DATA_BLOCK "InstCycleTimerDataset1"   // DB63
TITLE = Instanz CycleTimerDataset1 / Instance CycleTimerDataset1
{ DB_Accessible_From_OPC_UA := 'FALSE' }
AUTHOR : SICAR
FAMILY : ProdData
// Instanz DB / Instance DB
// stored: DBAccessibleFromOPCUA false, InstanceOfName LSicar_ProdDataCycleTimer, InstanceOfType FB
"LSicar_ProdDataCycleTimer"
   // VAR_INPUT
   //    numberConfigDataSets { ExternalAccessible := 'False'; ExternalVisible := 'False'; ExternalWritable := 'False'} : Int := 0;
   //    dataSetNumber { ExternalAccessible := 'False'; ExternalVisible := 'False'; ExternalWritable := 'False'} : UInt := 0;
   //    pulse100ms { ExternalAccessible := 'False'; ExternalVisible := 'False'; ExternalWritable := 'False'} : Bool := FALSE;
   // END_VAR
   // VAR_IN_OUT
   //    numberOfDataSets : "LSicar_typeNumberOfDataSets";
   //    dataSet : "LSicar_typeCycleTimer";
   // END_VAR
   // VAR
   //    statCycleTimer { ExternalAccessible := 'False'; ExternalVisible := 'False'; ExternalWritable := 'False'} : Array[0..20] of "LSicar_typeCycleTimerStruct";
   //    statRisEdgeResetAllExt { ExternalAccessible := 'False'; ExternalVisible := 'False'; ExternalWritable := 'False'} : Bool := FALSE;
   //    statPosPulseResetAllExt { ExternalAccessible := 'False'; ExternalVisible := 'False'; ExternalWritable := 'False'} : Bool := FALSE;
   //    statRisEdgeResetAll { ExternalAccessible := 'False'; ExternalVisible := 'False'; ExternalWritable := 'False'} : Bool := FALSE;
   //    statPosPulseResetAll { ExternalAccessible := 'False'; ExternalVisible := 'False'; ExternalWritable := 'False'} : Bool := FALSE;
   // END_VAR
BEGIN
   statCycleTimer[0..20].falEdgeRun := FALSE;
   statCycleTimer[0..20].negPulseRun := FALSE;
   statCycleTimer[0..20].risEdgeReset := FALSE;
   statCycleTimer[0..20].posPulseReset := FALSE;
   statCycleTimer[0..20].operateValue := 0;
END_DATA_BLOCK

DATA_BLOCK "InstCycleTimerDataset2"   // DB79
TITLE = Instanz CycleTimerDataset2 / Instance CycleTimerDataset2
{ DB_Accessible_From_OPC_UA := 'FALSE' }
AUTHOR : SICAR
FAMILY : ProdData
// Instanz DB / Instance DB
// stored: DBAccessibleFromOPCUA false, InstanceOfName LSicar_ProdDataCycleTimer, InstanceOfType FB
"LSicar_ProdDataCycleTimer"
   // VAR_INPUT
   //    numberConfigDataSets { ExternalAccessible := 'False'; ExternalVisible := 'False'; ExternalWritable := 'False'} : Int := 0;
   //    dataSetNumber { ExternalAccessible := 'False'; ExternalVisible := 'False'; ExternalWritable := 'False'} : UInt := 0;
   //    pulse100ms { ExternalAccessible := 'False'; ExternalVisible := 'False'; ExternalWritable := 'False'} : Bool := FALSE;
   // END_VAR
   // VAR_IN_OUT
   //    numberOfDataSets : "LSicar_typeNumberOfDataSets";
   //    dataSet : "LSicar_typeCycleTimer";
   // END_VAR
   // VAR
   //    statCycleTimer { ExternalAccessible := 'False'; ExternalVisible := 'False'; ExternalWritable := 'False'} : Array[0..20] of "LSicar_typeCycleTimerStruct";
   //    statRisEdgeResetAllExt { ExternalAccessible := 'False'; ExternalVisible := 'False'; ExternalWritable := 'False'} : Bool := FALSE;
   //    statPosPulseResetAllExt { ExternalAccessible := 'False'; ExternalVisible := 'False'; ExternalWritable := 'False'} : Bool := FALSE;
   //    statRisEdgeResetAll { ExternalAccessible := 'False'; ExternalVisible := 'False'; ExternalWritable := 'False'} : Bool := FALSE;
   //    statPosPulseResetAll { ExternalAccessible := 'False'; ExternalVisible := 'False'; ExternalWritable := 'False'} : Bool := FALSE;
   // END_VAR
BEGIN
   statCycleTimer[0..20].falEdgeRun := FALSE;
   statCycleTimer[0..20].negPulseRun := FALSE;
   statCycleTimer[0..20].risEdgeReset := FALSE;
   statCycleTimer[0..20].posPulseReset := FALSE;
   statCycleTimer[0..20].operateValue := 0;
END_DATA_BLOCK

DATA_BLOCK "InstCycleTimerDataset3"   // DB114
AUTHOR : SICAR
FAMILY : ProdData
VERSION : 1.0
// stored: InstanceOfName LSicar_ProdDataCycleTimer, InstanceOfType FB
"LSicar_ProdDataCycleTimer"
   // VAR_INPUT
   //    numberConfigDataSets { ExternalAccessible := 'False'; ExternalVisible := 'False'; ExternalWritable := 'False'} : Int;
   //    dataSetNumber { ExternalAccessible := 'False'; ExternalVisible := 'False'; ExternalWritable := 'False'} : UInt;
   //    pulse100ms { ExternalAccessible := 'False'; ExternalVisible := 'False'; ExternalWritable := 'False'} : Bool;
   // END_VAR
   // VAR_IN_OUT
   //    numberOfDataSets : "LSicar_typeNumberOfDataSets";
   //    dataSet : "LSicar_typeCycleTimer";
   // END_VAR
   // VAR
   //    statCycleTimer { ExternalAccessible := 'False'; ExternalVisible := 'False'; ExternalWritable := 'False'} : Array[0..20] of "LSicar_typeCycleTimerStruct";
   //    statRisEdgeResetAllExt { ExternalAccessible := 'False'; ExternalVisible := 'False'; ExternalWritable := 'False'} : Bool;
   //    statPosPulseResetAllExt { ExternalAccessible := 'False'; ExternalVisible := 'False'; ExternalWritable := 'False'} : Bool;
   //    statRisEdgeResetAll { ExternalAccessible := 'False'; ExternalVisible := 'False'; ExternalWritable := 'False'} : Bool;
   //    statPosPulseResetAll { ExternalAccessible := 'False'; ExternalVisible := 'False'; ExternalWritable := 'False'} : Bool;
   // END_VAR
BEGIN
END_DATA_BLOCK

DATA_BLOCK "InstCycleTimerDataset4"   // DB494
AUTHOR : SICAR
FAMILY : ProdData
VERSION : 1.0
// stored: InstanceOfName LSicar_ProdDataCycleTimer, InstanceOfType FB
"LSicar_ProdDataCycleTimer"
   // VAR_INPUT
   //    numberConfigDataSets { ExternalAccessible := 'False'; ExternalVisible := 'False'; ExternalWritable := 'False'} : Int;
   //    dataSetNumber { ExternalAccessible := 'False'; ExternalVisible := 'False'; ExternalWritable := 'False'} : UInt;
   //    pulse100ms { ExternalAccessible := 'False'; ExternalVisible := 'False'; ExternalWritable := 'False'} : Bool;
   // END_VAR
   // VAR_IN_OUT
   //    numberOfDataSets : "LSicar_typeNumberOfDataSets";
   //    dataSet : "LSicar_typeCycleTimer";
   // END_VAR
   // VAR
   //    statCycleTimer { ExternalAccessible := 'False'; ExternalVisible := 'False'; ExternalWritable := 'False'} : Array[0..20] of "LSicar_typeCycleTimerStruct";
   //    statRisEdgeResetAllExt { ExternalAccessible := 'False'; ExternalVisible := 'False'; ExternalWritable := 'False'} : Bool;
   //    statPosPulseResetAllExt { ExternalAccessible := 'False'; ExternalVisible := 'False'; ExternalWritable := 'False'} : Bool;
   //    statRisEdgeResetAll { ExternalAccessible := 'False'; ExternalVisible := 'False'; ExternalWritable := 'False'} : Bool;
   //    statPosPulseResetAll { ExternalAccessible := 'False'; ExternalVisible := 'False'; ExternalWritable := 'False'} : Bool;
   // END_VAR
BEGIN
END_DATA_BLOCK

DATA_BLOCK "InstCycleTimerDataset5"   // DB216
AUTHOR : SICAR
FAMILY : ProdData
VERSION : 1.0
// stored: InstanceOfName LSicar_ProdDataCycleTimer, InstanceOfType FB
"LSicar_ProdDataCycleTimer"
   // VAR_INPUT
   //    numberConfigDataSets { ExternalAccessible := 'False'; ExternalVisible := 'False'; ExternalWritable := 'False'} : Int;
   //    dataSetNumber { ExternalAccessible := 'False'; ExternalVisible := 'False'; ExternalWritable := 'False'} : UInt;
   //    pulse100ms { ExternalAccessible := 'False'; ExternalVisible := 'False'; ExternalWritable := 'False'} : Bool;
   // END_VAR
   // VAR_IN_OUT
   //    numberOfDataSets : "LSicar_typeNumberOfDataSets";
   //    dataSet : "LSicar_typeCycleTimer";
   // END_VAR
   // VAR
   //    statCycleTimer { ExternalAccessible := 'False'; ExternalVisible := 'False'; ExternalWritable := 'False'} : Array[0..20] of "LSicar_typeCycleTimerStruct";
   //    statRisEdgeResetAllExt { ExternalAccessible := 'False'; ExternalVisible := 'False'; ExternalWritable := 'False'} : Bool;
   //    statPosPulseResetAllExt { ExternalAccessible := 'False'; ExternalVisible := 'False'; ExternalWritable := 'False'} : Bool;
   //    statRisEdgeResetAll { ExternalAccessible := 'False'; ExternalVisible := 'False'; ExternalWritable := 'False'} : Bool;
   //    statPosPulseResetAll { ExternalAccessible := 'False'; ExternalVisible := 'False'; ExternalWritable := 'False'} : Bool;
   // END_VAR
BEGIN
END_DATA_BLOCK

DATA_BLOCK "InstCycleTimerDataset6"   // DB258
AUTHOR : SICAR
FAMILY : ProdData
VERSION : 1.0
// stored: InstanceOfName LSicar_ProdDataCycleTimer, InstanceOfType FB
"LSicar_ProdDataCycleTimer"
   // VAR_INPUT
   //    numberConfigDataSets { ExternalAccessible := 'False'; ExternalVisible := 'False'; ExternalWritable := 'False'} : Int;
   //    dataSetNumber { ExternalAccessible := 'False'; ExternalVisible := 'False'; ExternalWritable := 'False'} : UInt;
   //    pulse100ms { ExternalAccessible := 'False'; ExternalVisible := 'False'; ExternalWritable := 'False'} : Bool;
   // END_VAR
   // VAR_IN_OUT
   //    numberOfDataSets : "LSicar_typeNumberOfDataSets";
   //    dataSet : "LSicar_typeCycleTimer";
   // END_VAR
   // VAR
   //    statCycleTimer { ExternalAccessible := 'False'; ExternalVisible := 'False'; ExternalWritable := 'False'} : Array[0..20] of "LSicar_typeCycleTimerStruct";
   //    statRisEdgeResetAllExt { ExternalAccessible := 'False'; ExternalVisible := 'False'; ExternalWritable := 'False'} : Bool;
   //    statPosPulseResetAllExt { ExternalAccessible := 'False'; ExternalVisible := 'False'; ExternalWritable := 'False'} : Bool;
   //    statRisEdgeResetAll { ExternalAccessible := 'False'; ExternalVisible := 'False'; ExternalWritable := 'False'} : Bool;
   //    statPosPulseResetAll { ExternalAccessible := 'False'; ExternalVisible := 'False'; ExternalWritable := 'False'} : Bool;
   // END_VAR
BEGIN
END_DATA_BLOCK

DATA_BLOCK "InstCycleTimerDataset7"   // DB264
AUTHOR : SICAR
FAMILY : ProdData
VERSION : 1.0
// stored: InstanceOfName LSicar_ProdDataCycleTimer, InstanceOfType FB
"LSicar_ProdDataCycleTimer"
   // VAR_INPUT
   //    numberConfigDataSets { ExternalAccessible := 'False'; ExternalVisible := 'False'; ExternalWritable := 'False'} : Int;
   //    dataSetNumber { ExternalAccessible := 'False'; ExternalVisible := 'False'; ExternalWritable := 'False'} : UInt;
   //    pulse100ms { ExternalAccessible := 'False'; ExternalVisible := 'False'; ExternalWritable := 'False'} : Bool;
   // END_VAR
   // VAR_IN_OUT
   //    numberOfDataSets : "LSicar_typeNumberOfDataSets";
   //    dataSet : "LSicar_typeCycleTimer";
   // END_VAR
   // VAR
   //    statCycleTimer { ExternalAccessible := 'False'; ExternalVisible := 'False'; ExternalWritable := 'False'} : Array[0..20] of "LSicar_typeCycleTimerStruct";
   //    statRisEdgeResetAllExt { ExternalAccessible := 'False'; ExternalVisible := 'False'; ExternalWritable := 'False'} : Bool;
   //    statPosPulseResetAllExt { ExternalAccessible := 'False'; ExternalVisible := 'False'; ExternalWritable := 'False'} : Bool;
   //    statRisEdgeResetAll { ExternalAccessible := 'False'; ExternalVisible := 'False'; ExternalWritable := 'False'} : Bool;
   //    statPosPulseResetAll { ExternalAccessible := 'False'; ExternalVisible := 'False'; ExternalWritable := 'False'} : Bool;
   // END_VAR
BEGIN
END_DATA_BLOCK

DATA_BLOCK "InstCycleTimerDataset8"   // DB267
AUTHOR : SICAR
FAMILY : ProdData
VERSION : 1.0
// stored: InstanceOfName LSicar_ProdDataCycleTimer, InstanceOfType FB
"LSicar_ProdDataCycleTimer"
   // VAR_INPUT
   //    numberConfigDataSets { ExternalAccessible := 'False'; ExternalVisible := 'False'; ExternalWritable := 'False'} : Int;
   //    dataSetNumber { ExternalAccessible := 'False'; ExternalVisible := 'False'; ExternalWritable := 'False'} : UInt;
   //    pulse100ms { ExternalAccessible := 'False'; ExternalVisible := 'False'; ExternalWritable := 'False'} : Bool;
   // END_VAR
   // VAR_IN_OUT
   //    numberOfDataSets : "LSicar_typeNumberOfDataSets";
   //    dataSet : "LSicar_typeCycleTimer";
   // END_VAR
   // VAR
   //    statCycleTimer { ExternalAccessible := 'False'; ExternalVisible := 'False'; ExternalWritable := 'False'} : Array[0..20] of "LSicar_typeCycleTimerStruct";
   //    statRisEdgeResetAllExt { ExternalAccessible := 'False'; ExternalVisible := 'False'; ExternalWritable := 'False'} : Bool;
   //    statPosPulseResetAllExt { ExternalAccessible := 'False'; ExternalVisible := 'False'; ExternalWritable := 'False'} : Bool;
   //    statRisEdgeResetAll { ExternalAccessible := 'False'; ExternalVisible := 'False'; ExternalWritable := 'False'} : Bool;
   //    statPosPulseResetAll { ExternalAccessible := 'False'; ExternalVisible := 'False'; ExternalWritable := 'False'} : Bool;
   // END_VAR
BEGIN
END_DATA_BLOCK

DATA_BLOCK "InstLimitValueDataset1"   // DB54
TITLE = Instanz LimitValueDataset1 / Instance LimitValueDataset1
{ DB_Accessible_From_OPC_UA := 'FALSE' }
AUTHOR : SICAR
FAMILY : ProdData
// Instanz DB / Instance DB
// stored: DBAccessibleFromOPCUA false, InstanceOfName LSicar_ProdDataLimitValues, InstanceOfType FB
"LSicar_ProdDataLimitValues"
   // VAR_INPUT
   //    numberConfigDataSets { ExternalAccessible := 'False'; ExternalVisible := 'False'; ExternalWritable := 'False'} : Int := 0;
   //    dataSetNumber { ExternalAccessible := 'False'; ExternalVisible := 'False'; ExternalWritable := 'False'} : UInt := 0;
   // END_VAR
   // VAR_IN_OUT
   //    numberOfDataSets : "LSicar_typeNumberOfDataSets";
   //    dataSet : "LSicar_typeLimitValue";
   //    colorCodeSelectButton { ExternalAccessible := 'False'; ExternalVisible := 'False'; ExternalWritable := 'False'} : UInt := 0;
   // END_VAR
   // VAR
   //    statLimitValue { ExternalAccessible := 'False'; ExternalVisible := 'False'; ExternalWritable := 'False'} : Array[0..10] of "LSicar_typeEdgePulseStruct";
   //    statPrewarnActive { ExternalAccessible := 'False'; ExternalVisible := 'False'; ExternalWritable := 'False'} : Bool := FALSE;
   //    statAlarmActive { ExternalAccessible := 'False'; ExternalVisible := 'False'; ExternalWritable := 'False'} : Bool := FALSE;
   // END_VAR
BEGIN
   statLimitValue[0..10].risEdgeCountUp := FALSE;
   statLimitValue[0..10].posPulseCountUp := FALSE;
   statLimitValue[0..10].risEdgeCountDown := FALSE;
   statLimitValue[0..10].posPulseCountDown := FALSE;
   statLimitValue[0..10].risEdgeReset := FALSE;
   statLimitValue[0..10].posPulseReset := FALSE;
END_DATA_BLOCK

DATA_BLOCK "InstLimitValueDataset2"   // DB55
TITLE = Instanz LimitValueDataset2 / Instance LimitValueDataset2
{ DB_Accessible_From_OPC_UA := 'FALSE' }
AUTHOR : SICAR
FAMILY : ProdData
// Instanz DB / Instance DB
// stored: DBAccessibleFromOPCUA false, InstanceOfName LSicar_ProdDataLimitValues, InstanceOfType FB
"LSicar_ProdDataLimitValues"
   // VAR_INPUT
   //    numberConfigDataSets { ExternalAccessible := 'False'; ExternalVisible := 'False'; ExternalWritable := 'False'} : Int := 0;
   //    dataSetNumber { ExternalAccessible := 'False'; ExternalVisible := 'False'; ExternalWritable := 'False'} : UInt := 0;
   // END_VAR
   // VAR_IN_OUT
   //    numberOfDataSets : "LSicar_typeNumberOfDataSets";
   //    dataSet : "LSicar_typeLimitValue";
   //    colorCodeSelectButton { ExternalAccessible := 'False'; ExternalVisible := 'False'; ExternalWritable := 'False'} : UInt := 0;
   // END_VAR
   // VAR
   //    statLimitValue { ExternalAccessible := 'False'; ExternalVisible := 'False'; ExternalWritable := 'False'} : Array[0..10] of "LSicar_typeEdgePulseStruct";
   //    statPrewarnActive { ExternalAccessible := 'False'; ExternalVisible := 'False'; ExternalWritable := 'False'} : Bool := FALSE;
   //    statAlarmActive { ExternalAccessible := 'False'; ExternalVisible := 'False'; ExternalWritable := 'False'} : Bool := FALSE;
   // END_VAR
BEGIN
   statLimitValue[0..10].risEdgeCountUp := FALSE;
   statLimitValue[0..10].posPulseCountUp := FALSE;
   statLimitValue[0..10].risEdgeCountDown := FALSE;
   statLimitValue[0..10].posPulseCountDown := FALSE;
   statLimitValue[0..10].risEdgeReset := FALSE;
   statLimitValue[0..10].posPulseReset := FALSE;
END_DATA_BLOCK

DATA_BLOCK "InstShiftCounterDataset1"   // DB62
TITLE = Instanz ShiftCounterDataset1 / Instance ShiftCounterDataset1
{ DB_Accessible_From_OPC_UA := 'FALSE' }
AUTHOR : SICAR
FAMILY : ProdData
// Instanz DB / Instance DB
// stored: DBAccessibleFromOPCUA false, InstanceOfName LSicar_ProdDataShiftCounter, InstanceOfType FB
"LSicar_ProdDataShiftCounter"
   // VAR_INPUT
   //    numberConfigDataSets { ExternalAccessible := 'False'; ExternalVisible := 'False'; ExternalWritable := 'False'} : Int := 0;
   //    dataSetNumber { ExternalAccessible := 'False'; ExternalVisible := 'False'; ExternalWritable := 'False'} : UInt := 0;
   // END_VAR
   // VAR_IN_OUT
   //    numberOfDataSets : "LSicar_typeNumberOfDataSets";
   //    dataSet : "LSicar_typeShiftCounter";
   // END_VAR
   // VAR
   //    statPartsCurrentCount { ExternalAccessible := 'False'; ExternalVisible := 'False'; ExternalWritable := 'False'} : Array[0..10] of "LSicar_typeEdgePulseStruct";
   //    statRisEdgeResetAllExt { ExternalAccessible := 'False'; ExternalVisible := 'False'; ExternalWritable := 'False'} : Bool := FALSE;
   //    statPosPulseResetAllExt { ExternalAccessible := 'False'; ExternalVisible := 'False'; ExternalWritable := 'False'} : Bool := FALSE;
   //    statRisEdgeResetAll { ExternalAccessible := 'False'; ExternalVisible := 'False'; ExternalWritable := 'False'} : Bool := FALSE;
   //    statPosPulseResetAll { ExternalAccessible := 'False'; ExternalVisible := 'False'; ExternalWritable := 'False'} : Bool := FALSE;
   // END_VAR
BEGIN
   statPartsCurrentCount[0..10].risEdgeCountUp := FALSE;
   statPartsCurrentCount[0..10].posPulseCountUp := FALSE;
   statPartsCurrentCount[0..10].risEdgeCountDown := FALSE;
   statPartsCurrentCount[0..10].posPulseCountDown := FALSE;
   statPartsCurrentCount[0..10].risEdgeReset := FALSE;
   statPartsCurrentCount[0..10].posPulseReset := FALSE;
END_DATA_BLOCK

DATA_BLOCK "InstShiftCounterDataset2"   // DB64
TITLE = Instanz ShiftCounterDataset2 / Instance ShiftCounterDataset2
{ DB_Accessible_From_OPC_UA := 'FALSE' }
AUTHOR : SICAR
FAMILY : ProdData
// Instanz DB / Instance DB
// stored: DBAccessibleFromOPCUA false, InstanceOfName LSicar_ProdDataShiftCounter, InstanceOfType FB
"LSicar_ProdDataShiftCounter"
   // VAR_INPUT
   //    numberConfigDataSets { ExternalAccessible := 'False'; ExternalVisible := 'False'; ExternalWritable := 'False'} : Int := 0;
   //    dataSetNumber { ExternalAccessible := 'False'; ExternalVisible := 'False'; ExternalWritable := 'False'} : UInt := 0;
   // END_VAR
   // VAR_IN_OUT
   //    numberOfDataSets : "LSicar_typeNumberOfDataSets";
   //    dataSet : "LSicar_typeShiftCounter";
   // END_VAR
   // VAR
   //    statPartsCurrentCount { ExternalAccessible := 'False'; ExternalVisible := 'False'; ExternalWritable := 'False'} : Array[0..10] of "LSicar_typeEdgePulseStruct";
   //    statRisEdgeResetAllExt { ExternalAccessible := 'False'; ExternalVisible := 'False'; ExternalWritable := 'False'} : Bool := FALSE;
   //    statPosPulseResetAllExt { ExternalAccessible := 'False'; ExternalVisible := 'False'; ExternalWritable := 'False'} : Bool := FALSE;
   //    statRisEdgeResetAll { ExternalAccessible := 'False'; ExternalVisible := 'False'; ExternalWritable := 'False'} : Bool := FALSE;
   //    statPosPulseResetAll { ExternalAccessible := 'False'; ExternalVisible := 'False'; ExternalWritable := 'False'} : Bool := FALSE;
   // END_VAR
BEGIN
   statPartsCurrentCount[0..10].risEdgeCountUp := FALSE;
   statPartsCurrentCount[0..10].posPulseCountUp := FALSE;
   statPartsCurrentCount[0..10].risEdgeCountDown := FALSE;
   statPartsCurrentCount[0..10].posPulseCountDown := FALSE;
   statPartsCurrentCount[0..10].risEdgeReset := FALSE;
   statPartsCurrentCount[0..10].posPulseReset := FALSE;
END_DATA_BLOCK

DATA_BLOCK "InstShiftCounterOeeDset1"   // DB124
TITLE = Instanz ShiftCounterOeeDset1 / Instance ShiftCounterOeeDset1
{ DB_Accessible_From_OPC_UA := 'FALSE' }
AUTHOR : SICAR
FAMILY : ProdData
// Instanz DB / Instance DB
// stored: DBAccessibleFromOPCUA false, InstanceOfName LSicar_ProdDataShiftCounterOee, InstanceOfType FB
"LSicar_ProdDataShiftCounterOee"
   // VAR_INPUT
   //    numberConfigDataSets { ExternalAccessible := 'False'; ExternalVisible := 'False'; ExternalWritable := 'False'} : Int := 0;
   //    dataSetNumber { ExternalAccessible := 'False'; ExternalVisible := 'False'; ExternalWritable := 'False'} : UInt := 0;
   //    shiftProdTimeTarget { ExternalAccessible := 'False'; ExternalVisible := 'False'; ExternalWritable := 'False'} : Time := T#0MS;
   //    shiftProdTimeExpired { ExternalAccessible := 'False'; ExternalVisible := 'False'; ExternalWritable := 'False'} : Time := T#0MS;
   // END_VAR
   // VAR_IN_OUT
   //    numberOfDataSets : "LSicar_typeNumberOfDataSets";
   //    dataSet : "LSicar_typeShiftCounterOee";
   // END_VAR
   // VAR
   //    statPartsCurrentCount { ExternalAccessible := 'False'; ExternalVisible := 'False'; ExternalWritable := 'False'} : Array[0..10] of "LSicar_typeEdgePulseStruct";
   //    statPartsCurrentCountOk { ExternalAccessible := 'False'; ExternalVisible := 'False'; ExternalWritable := 'False'} : Array[0..10] of "LSicar_typeEdgePulseStruct";
   //    statFactor { ExternalAccessible := 'False'; ExternalVisible := 'False'; ExternalWritable := 'False'} : "LSicar_typeFactorOee";
   //    statTimeFactorTrend { ExternalAccessible := 'False'; ExternalVisible := 'False'; ExternalWritable := 'False'} : Real := 0.0;
   //    statShiftProdTimeTarget { ExternalAccessible := 'False'; ExternalVisible := 'False'; ExternalWritable := 'False'} : Real := 0.0;
   //    statShiftProdTimeExpired { ExternalAccessible := 'False'; ExternalVisible := 'False'; ExternalWritable := 'False'} : Real := 0.0;
   //    statRisEdgeResetAllExt { ExternalAccessible := 'False'; ExternalVisible := 'False'; ExternalWritable := 'False'} : Bool := FALSE;
   //    statPosPulseResetAllExt { ExternalAccessible := 'False'; ExternalVisible := 'False'; ExternalWritable := 'False'} : Bool := FALSE;
   //    statRisEdgeResetAll { ExternalAccessible := 'False'; ExternalVisible := 'False'; ExternalWritable := 'False'} : Bool := FALSE;
   //    statPosPulseResetAll { ExternalAccessible := 'False'; ExternalVisible := 'False'; ExternalWritable := 'False'} : Bool := FALSE;
   // END_VAR
BEGIN
   statPartsCurrentCount[0..10].risEdgeCountUp := FALSE;
   statPartsCurrentCount[0..10].posPulseCountUp := FALSE;
   statPartsCurrentCount[0..10].risEdgeCountDown := FALSE;
   statPartsCurrentCount[0..10].posPulseCountDown := FALSE;
   statPartsCurrentCount[0..10].risEdgeReset := FALSE;
   statPartsCurrentCount[0..10].posPulseReset := FALSE;
   statPartsCurrentCountOk[0..10].risEdgeCountUp := FALSE;
   statPartsCurrentCountOk[0..10].posPulseCountUp := FALSE;
   statPartsCurrentCountOk[0..10].risEdgeCountDown := FALSE;
   statPartsCurrentCountOk[0..10].posPulseCountDown := FALSE;
   statPartsCurrentCountOk[0..10].risEdgeReset := FALSE;
   statPartsCurrentCountOk[0..10].posPulseReset := FALSE;
   statFactor.utilization := 0.0;
   statFactor.efficiency := 0.0;
   statFactor.quality := 0.0;
END_DATA_BLOCK

DATA_BLOCK "InstShiftCounterOeeDset2"   // DB125
TITLE = Instanz ShiftCounterOeeDset2 / Instance ShiftCounterOeeDset2
{ DB_Accessible_From_OPC_UA := 'FALSE' }
AUTHOR : SICAR
FAMILY : ProdData
// Instanz DB / Instance DB
// stored: DBAccessibleFromOPCUA false, InstanceOfName LSicar_ProdDataShiftCounterOee, InstanceOfType FB
"LSicar_ProdDataShiftCounterOee"
   // VAR_INPUT
   //    numberConfigDataSets { ExternalAccessible := 'False'; ExternalVisible := 'False'; ExternalWritable := 'False'} : Int := 0;
   //    dataSetNumber { ExternalAccessible := 'False'; ExternalVisible := 'False'; ExternalWritable := 'False'} : UInt := 0;
   //    shiftProdTimeTarget { ExternalAccessible := 'False'; ExternalVisible := 'False'; ExternalWritable := 'False'} : Time := T#0MS;
   //    shiftProdTimeExpired { ExternalAccessible := 'False'; ExternalVisible := 'False'; ExternalWritable := 'False'} : Time := T#0MS;
   // END_VAR
   // VAR_IN_OUT
   //    numberOfDataSets : "LSicar_typeNumberOfDataSets";
   //    dataSet : "LSicar_typeShiftCounterOee";
   // END_VAR
   // VAR
   //    statPartsCurrentCount { ExternalAccessible := 'False'; ExternalVisible := 'False'; ExternalWritable := 'False'} : Array[0..10] of "LSicar_typeEdgePulseStruct";
   //    statPartsCurrentCountOk { ExternalAccessible := 'False'; ExternalVisible := 'False'; ExternalWritable := 'False'} : Array[0..10] of "LSicar_typeEdgePulseStruct";
   //    statFactor { ExternalAccessible := 'False'; ExternalVisible := 'False'; ExternalWritable := 'False'} : "LSicar_typeFactorOee";
   //    statTimeFactorTrend { ExternalAccessible := 'False'; ExternalVisible := 'False'; ExternalWritable := 'False'} : Real := 0.0;
   //    statShiftProdTimeTarget { ExternalAccessible := 'False'; ExternalVisible := 'False'; ExternalWritable := 'False'} : Real := 0.0;
   //    statShiftProdTimeExpired { ExternalAccessible := 'False'; ExternalVisible := 'False'; ExternalWritable := 'False'} : Real := 0.0;
   //    statRisEdgeResetAllExt { ExternalAccessible := 'False'; ExternalVisible := 'False'; ExternalWritable := 'False'} : Bool := FALSE;
   //    statPosPulseResetAllExt { ExternalAccessible := 'False'; ExternalVisible := 'False'; ExternalWritable := 'False'} : Bool := FALSE;
   //    statRisEdgeResetAll { ExternalAccessible := 'False'; ExternalVisible := 'False'; ExternalWritable := 'False'} : Bool := FALSE;
   //    statPosPulseResetAll { ExternalAccessible := 'False'; ExternalVisible := 'False'; ExternalWritable := 'False'} : Bool := FALSE;
   // END_VAR
BEGIN
   statPartsCurrentCount[0..10].risEdgeCountUp := FALSE;
   statPartsCurrentCount[0..10].posPulseCountUp := FALSE;
   statPartsCurrentCount[0..10].risEdgeCountDown := FALSE;
   statPartsCurrentCount[0..10].posPulseCountDown := FALSE;
   statPartsCurrentCount[0..10].risEdgeReset := FALSE;
   statPartsCurrentCount[0..10].posPulseReset := FALSE;
   statPartsCurrentCountOk[0..10].risEdgeCountUp := FALSE;
   statPartsCurrentCountOk[0..10].posPulseCountUp := FALSE;
   statPartsCurrentCountOk[0..10].risEdgeCountDown := FALSE;
   statPartsCurrentCountOk[0..10].posPulseCountDown := FALSE;
   statPartsCurrentCountOk[0..10].risEdgeReset := FALSE;
   statPartsCurrentCountOk[0..10].posPulseReset := FALSE;
   statFactor.utilization := 0.0;
   statFactor.efficiency := 0.0;
   statFactor.quality := 0.0;
END_DATA_BLOCK

DATA_BLOCK "InstShiftProductionTimes"   // DB113
TITLE = Instance ShiftProductionTimes
{ DB_Accessible_From_OPC_UA := 'FALSE' }
AUTHOR : SICAR
FAMILY : Shift
// Instance DB
// stored: DBAccessibleFromOPCUA false, InstanceOfName LSicar_ShiftProductionTimes, InstanceOfType FB
"LSicar_ShiftProductionTimes"
   // VAR_OUTPUT
   //    shiftProdTimeTarget { ExternalAccessible := 'False'; ExternalVisible := 'False'; ExternalWritable := 'False'} : Time := T#0MS;
   //    shiftProdTimeExpired { ExternalAccessible := 'False'; ExternalVisible := 'False'; ExternalWritable := 'False'} : Time := T#0MS;
   //    shiftActive { ExternalAccessible := 'False'; ExternalVisible := 'False'; ExternalWritable := 'False'} : Bool := FALSE;
   //    shiftFinishedPulse { ExternalAccessible := 'False'; ExternalVisible := 'False'; ExternalWritable := 'False'} : Bool := FALSE;
   // END_VAR
   // VAR_IN_OUT
   //    dateAndTime : "LSicar_typeGlobalDateTime";
   //    prodTimesHmi : "LSicar_typeProdTimesHmi";
   // END_VAR
   // VAR
   //    statCurrShiftTimes { ExternalAccessible := 'False'; ExternalVisible := 'False'; ExternalWritable := 'False'} : "LSicar_typeShiftTimes1Shift";
   //    statActual { ExternalAccessible := 'False'; ExternalVisible := 'False'; ExternalWritable := 'False'} : Time_Of_Day := TOD#00:00:00;
   //    statBefore { ExternalAccessible := 'False'; ExternalVisible := 'False'; ExternalWritable := 'False'} : Time_Of_Day := TOD#00:00:00;
   //    statDayChange { ExternalAccessible := 'False'; ExternalVisible := 'False'; ExternalWritable := 'False'} : Bool := FALSE;
   //    statDayChangeSet { ExternalAccessible := 'False'; ExternalVisible := 'False'; ExternalWritable := 'False'} : Bool := FALSE;
   //    statShift { ExternalAccessible := 'False'; ExternalVisible := 'False'; ExternalWritable := 'False'} : "LSicar_typeShiftmodelInfo";
   //    statProdTimeExpired { ExternalAccessible := 'False'; ExternalVisible := 'False'; ExternalWritable := 'False'} : Time := T#0MS;
   //    statBreak { ExternalAccessible := 'False'; ExternalVisible := 'False'; ExternalWritable := 'False'} : Array[0..4] of "LSicar_typeShiftmodelInfo";
   //    statBreakDurationSummary { ExternalAccessible := 'False'; ExternalVisible := 'False'; ExternalWritable := 'False'} : Time := T#0MS;
   //    statBreakActiveSummary { ExternalAccessible := 'False'; ExternalVisible := 'False'; ExternalWritable := 'False'} : Bool := FALSE;
   //    statBreakCount { ExternalAccessible := 'False'; ExternalVisible := 'False'; ExternalWritable := 'False'} : USInt := 0;
   //    statProdTimeExpired1 { ExternalAccessible := 'False'; ExternalVisible := 'False'; ExternalWritable := 'False'} : Time := T#0MS;
   //    statProdTimeExpired2 { ExternalAccessible := 'False'; ExternalVisible := 'False'; ExternalWritable := 'False'} : Time := T#0MS;
   //    statFalEdgeShiftActive { ExternalAccessible := 'False'; ExternalVisible := 'False'; ExternalWritable := 'False'} : Bool := FALSE;
   //    statNegPulseShiftActive { ExternalAccessible := 'False'; ExternalVisible := 'False'; ExternalWritable := 'False'} : Bool := FALSE;
   // END_VAR
BEGIN
   statCurrShiftTimes.start := TOD#00:00:00;
   statCurrShiftTimes.break[0..4].start := TOD#00:00:00;
   statCurrShiftTimes.break[0..4].startCircuitTime := TOD#00:00:00;
   statCurrShiftTimes.break[0..4].endCircuitTime := TOD#00:00:00;
   statCurrShiftTimes.break[0..4].end := TOD#00:00:00;
   statCurrShiftTimes.end := TOD#00:00:00;
   statShift.configured := FALSE;
   statShift.active := FALSE;
   statShift.duration := T#0MS;
   statBreak[0..4].configured := FALSE;
   statBreak[0..4].active := FALSE;
   statBreak[0..4].duration := T#0MS;
END_DATA_BLOCK

DATA_BLOCK "InstShiftmodel"   // DB101
TITLE = Instanz Shiftmodel / InstanceShiftmodel
{ DB_Accessible_From_OPC_UA := 'FALSE' }
AUTHOR : SICAR
FAMILY : Shiftmodel
// Instanz DB / Instance DB
// stored: DBAccessibleFromOPCUA false, InstanceOfName LSicar_Shiftmodel, InstanceOfType FB
"LSicar_Shiftmodel"
   // VAR_OUTPUT
   //    currentShiftCircuitTimes { ExternalAccessible := 'False'; ExternalVisible := 'False'; ExternalWritable := 'False'} : "LSicar_typeShiftmodTime1Shift";
   //    currentShiftTimes { ExternalAccessible := 'False'; ExternalVisible := 'False'; ExternalWritable := 'False'} : "LSicar_typeShiftTimes1Shift";
   // END_VAR
   // VAR_IN_OUT
   //    dateAndTime : "LSicar_typeGlobalDateTime";
   //    shiftTimesHmi : "LSicar_typeShiftmodelHmi";
   //    shiftTimesList : Array[0..10] of "LSicar_typeShiftmodTime1DaySel";
   // END_VAR
   // VAR
   //    statListIdx { ExternalAccessible := 'False'; ExternalVisible := 'False'; ExternalWritable := 'False'} : DInt := 0;
   //    statHmiTimesDay { ExternalAccessible := 'False'; ExternalVisible := 'False'; ExternalWritable := 'False'} : Array[0..7] of "LSicar_typeShiftmodTime1Day";
   //    statHmiSignalsDay { ExternalAccessible := 'False'; ExternalVisible := 'False'; ExternalWritable := 'False'} : Array[0..7] of "LSicar_typeShiftmodSign1Day";
   //    statHmiActualDay { ExternalAccessible := 'False'; ExternalVisible := 'False'; ExternalWritable := 'False'} : USInt := 0;
   //    statShiftTimesListOn { ExternalAccessible := 'False'; ExternalVisible := 'False'; ExternalWritable := 'False'} : Bool := FALSE;
   //    statSummaryHmi { ExternalAccessible := 'False'; ExternalVisible := 'False'; ExternalWritable := 'False'} : "LSicar_typeShiftmodSumHmi";
   //    statHmiShiftmoListindex { ExternalAccessible := 'False'; ExternalVisible := 'False'; ExternalWritable := 'False'} : USInt := 1;
   //    statZeroDay { ExternalAccessible := 'False'; ExternalVisible := 'False'; ExternalWritable := 'False'} : "LSicar_typeShiftmodTime1Day";
   //    statListIndexOld { ExternalAccessible := 'False'; ExternalVisible := 'False'; ExternalWritable := 'False'} : DInt := 1;
   //    statNumberOfWorkDays { ExternalAccessible := 'False'; ExternalVisible := 'False'; ExternalWritable := 'False'} : USInt := 0;
   //    statTimeOfDayActual { ExternalAccessible := 'False'; ExternalVisible := 'False'; ExternalWritable := 'False'} : Time_Of_Day := TOD#00:00:00;
   //    statShiftActual { ExternalAccessible := 'False'; ExternalVisible := 'False'; ExternalWritable := 'False'} : USInt := 0;
   //    statDayCount { ExternalAccessible := 'False'; ExternalVisible := 'False'; ExternalWritable := 'False'} : USInt := 1;
   //    statBreakCount { ExternalAccessible := 'False'; ExternalVisible := 'False'; ExternalWritable := 'False'} : USInt := 0;
   //    statDayChangeNightShift { ExternalAccessible := 'False'; ExternalVisible := 'False'; ExternalWritable := 'False'} : Bool := FALSE;
   //    statDayChangeCircuitTime { ExternalAccessible := 'False'; ExternalVisible := 'False'; ExternalWritable := 'False'} : Bool := FALSE;
   //    statCheckCircuitTime { ExternalAccessible := 'False'; ExternalVisible := 'False'; ExternalWritable := 'False'} : "LSicar_typeShiftCircuitTimes";
   //    statRisEdge { ExternalAccessible := 'False'; ExternalVisible := 'False'; ExternalWritable := 'False'} : "LSicar_typeShiftmodSumHmi";
   //    statPosPulse { ExternalAccessible := 'False'; ExternalVisible := 'False'; ExternalWritable := 'False'} : "LSicar_typeShiftmodSumHmi";
   //    statFalEdge { ExternalAccessible := 'False'; ExternalVisible := 'False'; ExternalWritable := 'False'} : "LSicar_typeShiftmodSumHmi";
   //    statNegPulse { ExternalAccessible := 'False'; ExternalVisible := 'False'; ExternalWritable := 'False'} : "LSicar_typeShiftmodSumHmi";
   //    statTimesAndCircuit { ExternalAccessible := 'False'; ExternalVisible := 'False'; ExternalWritable := 'False'} : "LSicar_typeShiftmodTime1Shift";
   //    statOnlyTimes { ExternalAccessible := 'False'; ExternalVisible := 'False'; ExternalWritable := 'False'} : "LSicar_typeShiftTimes1Shift";
   //    statRisEdgeListOn { ExternalAccessible := 'False'; ExternalVisible := 'False'; ExternalWritable := 'False'} : Bool := FALSE;
   //    statPosPulseListOn { ExternalAccessible := 'False'; ExternalVisible := 'False'; ExternalWritable := 'False'} : Bool := FALSE;
   //    statFalEdgeListOn { ExternalAccessible := 'False'; ExternalVisible := 'False'; ExternalWritable := 'False'} : Bool := FALSE;
   //    statNegPulseListOn { ExternalAccessible := 'False'; ExternalVisible := 'False'; ExternalWritable := 'False'} : Bool := FALSE;
   //    statRisEdgeListChange { ExternalAccessible := 'False'; ExternalVisible := 'False'; ExternalWritable := 'False'} : Bool := FALSE;
   //    statPosPulseListChange { ExternalAccessible := 'False'; ExternalVisible := 'False'; ExternalWritable := 'False'} : Bool := FALSE;
   //    statFirstCycle { ExternalAccessible := 'False'; ExternalVisible := 'False'; ExternalWritable := 'False'} : Bool := TRUE;
   // END_VAR
BEGIN
   currentShiftCircuitTimes.endCircuitTime := TOD#00:00:00;
   currentShiftCircuitTimes.start := TOD#00:00:00;
   currentShiftCircuitTimes.break[0..4].start := TOD#00:00:00;
   currentShiftCircuitTimes.break[0..4].startCircuitTime := TOD#00:00:00;
   currentShiftCircuitTimes.break[0..4].endCircuitTime := TOD#00:00:00;
   currentShiftCircuitTimes.break[0..4].end := TOD#00:00:00;
   currentShiftCircuitTimes.end := TOD#00:00:00;
   currentShiftCircuitTimes.startCircuitTime := TOD#00:00:00;
   currentShiftTimes.start := TOD#00:00:00;
   currentShiftTimes.break[0..4].start := TOD#00:00:00;
   currentShiftTimes.break[0..4].startCircuitTime := TOD#00:00:00;
   currentShiftTimes.break[0..4].endCircuitTime := TOD#00:00:00;
   currentShiftTimes.break[0..4].end := TOD#00:00:00;
   currentShiftTimes.end := TOD#00:00:00;
   statHmiTimesDay[0].shift[0..3].endCircuitTime := TOD#00:00:00;
   statHmiTimesDay[1].shift[0..3].endCircuitTime := TOD#00:00:00;
   statHmiTimesDay[2].shift[0..3].endCircuitTime := TOD#00:00:00;
   statHmiTimesDay[3].shift[0..3].endCircuitTime := TOD#00:00:00;
   statHmiTimesDay[4].shift[0..3].endCircuitTime := TOD#00:00:00;
   statHmiTimesDay[5].shift[0..3].endCircuitTime := TOD#00:00:00;
   statHmiTimesDay[6].shift[0..3].endCircuitTime := TOD#00:00:00;
   statHmiTimesDay[7].shift[0..3].endCircuitTime := TOD#00:00:00;
   statHmiTimesDay[0].shift[0..3].start := TOD#00:00:00;
   statHmiTimesDay[1].shift[0..3].start := TOD#00:00:00;
   statHmiTimesDay[2].shift[0..3].start := TOD#00:00:00;
   statHmiTimesDay[3].shift[0..3].start := TOD#00:00:00;
   statHmiTimesDay[4].shift[0..3].start := TOD#00:00:00;
   statHmiTimesDay[5].shift[0..3].start := TOD#00:00:00;
   statHmiTimesDay[6].shift[0..3].start := TOD#00:00:00;
   statHmiTimesDay[7].shift[0..3].start := TOD#00:00:00;
   statHmiTimesDay[0].shift[0].break[0..4].start := TOD#00:00:00;
   statHmiTimesDay[0].shift[1].break[0..4].start := TOD#00:00:00;
   statHmiTimesDay[0].shift[2].break[0..4].start := TOD#00:00:00;
   statHmiTimesDay[0].shift[3].break[0..4].start := TOD#00:00:00;
   statHmiTimesDay[1].shift[0].break[0..4].start := TOD#00:00:00;
   statHmiTimesDay[1].shift[1].break[0..4].start := TOD#00:00:00;
   statHmiTimesDay[1].shift[2].break[0..4].start := TOD#00:00:00;
   statHmiTimesDay[1].shift[3].break[0..4].start := TOD#00:00:00;
   statHmiTimesDay[2].shift[0].break[0..4].start := TOD#00:00:00;
   statHmiTimesDay[2].shift[1].break[0..4].start := TOD#00:00:00;
   statHmiTimesDay[2].shift[2].break[0..4].start := TOD#00:00:00;
   statHmiTimesDay[2].shift[3].break[0..4].start := TOD#00:00:00;
   statHmiTimesDay[3].shift[0].break[0..4].start := TOD#00:00:00;
   statHmiTimesDay[3].shift[1].break[0..4].start := TOD#00:00:00;
   statHmiTimesDay[3].shift[2].break[0..4].start := TOD#00:00:00;
   statHmiTimesDay[3].shift[3].break[0..4].start := TOD#00:00:00;
   statHmiTimesDay[4].shift[0].break[0..4].start := TOD#00:00:00;
   statHmiTimesDay[4].shift[1].break[0..4].start := TOD#00:00:00;
   statHmiTimesDay[4].shift[2].break[0..4].start := TOD#00:00:00;
   statHmiTimesDay[4].shift[3].break[0..4].start := TOD#00:00:00;
   statHmiTimesDay[5].shift[0].break[0..4].start := TOD#00:00:00;
   statHmiTimesDay[5].shift[1].break[0..4].start := TOD#00:00:00;
   statHmiTimesDay[5].shift[2].break[0..4].start := TOD#00:00:00;
   statHmiTimesDay[5].shift[3].break[0..4].start := TOD#00:00:00;
   statHmiTimesDay[6].shift[0].break[0..4].start := TOD#00:00:00;
   statHmiTimesDay[6].shift[1].break[0..4].start := TOD#00:00:00;
   statHmiTimesDay[6].shift[2].break[0..4].start := TOD#00:00:00;
   statHmiTimesDay[6].shift[3].break[0..4].start := TOD#00:00:00;
   statHmiTimesDay[7].shift[0].break[0..4].start := TOD#00:00:00;
   statHmiTimesDay[7].shift[1].break[0..4].start := TOD#00:00:00;
   statHmiTimesDay[7].shift[2].break[0..4].start := TOD#00:00:00;
   statHmiTimesDay[7].shift[3].break[0..4].start := TOD#00:00:00;
   statHmiTimesDay[0].shift[0].break[0..4].startCircuitTime := TOD#00:00:00;
   statHmiTimesDay[0].shift[1].break[0..4].startCircuitTime := TOD#00:00:00;
   statHmiTimesDay[0].shift[2].break[0..4].startCircuitTime := TOD#00:00:00;
   statHmiTimesDay[0].shift[3].break[0..4].startCircuitTime := TOD#00:00:00;
   statHmiTimesDay[1].shift[0].break[0..4].startCircuitTime := TOD#00:00:00;
   statHmiTimesDay[1].shift[1].break[0..4].startCircuitTime := TOD#00:00:00;
   statHmiTimesDay[1].shift[2].break[0..4].startCircuitTime := TOD#00:00:00;
   statHmiTimesDay[1].shift[3].break[0..4].startCircuitTime := TOD#00:00:00;
   statHmiTimesDay[2].shift[0].break[0..4].startCircuitTime := TOD#00:00:00;
   statHmiTimesDay[2].shift[1].break[0..4].startCircuitTime := TOD#00:00:00;
   statHmiTimesDay[2].shift[2].break[0..4].startCircuitTime := TOD#00:00:00;
   statHmiTimesDay[2].shift[3].break[0..4].startCircuitTime := TOD#00:00:00;
   statHmiTimesDay[3].shift[0].break[0..4].startCircuitTime := TOD#00:00:00;
   statHmiTimesDay[3].shift[1].break[0..4].startCircuitTime := TOD#00:00:00;
   statHmiTimesDay[3].shift[2].break[0..4].startCircuitTime := TOD#00:00:00;
   statHmiTimesDay[3].shift[3].break[0..4].startCircuitTime := TOD#00:00:00;
   statHmiTimesDay[4].shift[0].break[0..4].startCircuitTime := TOD#00:00:00;
   statHmiTimesDay[4].shift[1].break[0..4].startCircuitTime := TOD#00:00:00;
   statHmiTimesDay[4].shift[2].break[0..4].startCircuitTime := TOD#00:00:00;
   statHmiTimesDay[4].shift[3].break[0..4].startCircuitTime := TOD#00:00:00;
   statHmiTimesDay[5].shift[0].break[0..4].startCircuitTime := TOD#00:00:00;
   statHmiTimesDay[5].shift[1].break[0..4].startCircuitTime := TOD#00:00:00;
   statHmiTimesDay[5].shift[2].break[0..4].startCircuitTime := TOD#00:00:00;
   statHmiTimesDay[5].shift[3].break[0..4].startCircuitTime := TOD#00:00:00;
   statHmiTimesDay[6].shift[0].break[0..4].startCircuitTime := TOD#00:00:00;
   statHmiTimesDay[6].shift[1].break[0..4].startCircuitTime := TOD#00:00:00;
   statHmiTimesDay[6].shift[2].break[0..4].startCircuitTime := TOD#00:00:00;
   statHmiTimesDay[6].shift[3].break[0..4].startCircuitTime := TOD#00:00:00;
   statHmiTimesDay[7].shift[0].break[0..4].startCircuitTime := TOD#00:00:00;
   statHmiTimesDay[7].shift[1].break[0..4].startCircuitTime := TOD#00:00:00;
   statHmiTimesDay[7].shift[2].break[0..4].startCircuitTime := TOD#00:00:00;
   statHmiTimesDay[7].shift[3].break[0..4].startCircuitTime := TOD#00:00:00;
   statHmiTimesDay[0].shift[0].break[0..4].endCircuitTime := TOD#00:00:00;
   statHmiTimesDay[0].shift[1].break[0..4].endCircuitTime := TOD#00:00:00;
   statHmiTimesDay[0].shift[2].break[0..4].endCircuitTime := TOD#00:00:00;
   statHmiTimesDay[0].shift[3].break[0..4].endCircuitTime := TOD#00:00:00;
   statHmiTimesDay[1].shift[0].break[0..4].endCircuitTime := TOD#00:00:00;
   statHmiTimesDay[1].shift[1].break[0..4].endCircuitTime := TOD#00:00:00;
   statHmiTimesDay[1].shift[2].break[0..4].endCircuitTime := TOD#00:00:00;
   statHmiTimesDay[1].shift[3].break[0..4].endCircuitTime := TOD#00:00:00;
   statHmiTimesDay[2].shift[0].break[0..4].endCircuitTime := TOD#00:00:00;
   statHmiTimesDay[2].shift[1].break[0..4].endCircuitTime := TOD#00:00:00;
   statHmiTimesDay[2].shift[2].break[0..4].endCircuitTime := TOD#00:00:00;
   statHmiTimesDay[2].shift[3].break[0..4].endCircuitTime := TOD#00:00:00;
   statHmiTimesDay[3].shift[0].break[0..4].endCircuitTime := TOD#00:00:00;
   statHmiTimesDay[3].shift[1].break[0..4].endCircuitTime := TOD#00:00:00;
   statHmiTimesDay[3].shift[2].break[0..4].endCircuitTime := TOD#00:00:00;
   statHmiTimesDay[3].shift[3].break[0..4].endCircuitTime := TOD#00:00:00;
   statHmiTimesDay[4].shift[0].break[0..4].endCircuitTime := TOD#00:00:00;
   statHmiTimesDay[4].shift[1].break[0..4].endCircuitTime := TOD#00:00:00;
   statHmiTimesDay[4].shift[2].break[0..4].endCircuitTime := TOD#00:00:00;
   statHmiTimesDay[4].shift[3].break[0..4].endCircuitTime := TOD#00:00:00;
   statHmiTimesDay[5].shift[0].break[0..4].endCircuitTime := TOD#00:00:00;
   statHmiTimesDay[5].shift[1].break[0..4].endCircuitTime := TOD#00:00:00;
   statHmiTimesDay[5].shift[2].break[0..4].endCircuitTime := TOD#00:00:00;
   statHmiTimesDay[5].shift[3].break[0..4].endCircuitTime := TOD#00:00:00;
   statHmiTimesDay[6].shift[0].break[0..4].endCircuitTime := TOD#00:00:00;
   statHmiTimesDay[6].shift[1].break[0..4].endCircuitTime := TOD#00:00:00;
   statHmiTimesDay[6].shift[2].break[0..4].endCircuitTime := TOD#00:00:00;
   statHmiTimesDay[6].shift[3].break[0..4].endCircuitTime := TOD#00:00:00;
   statHmiTimesDay[7].shift[0].break[0..4].endCircuitTime := TOD#00:00:00;
   statHmiTimesDay[7].shift[1].break[0..4].endCircuitTime := TOD#00:00:00;
   statHmiTimesDay[7].shift[2].break[0..4].endCircuitTime := TOD#00:00:00;
   statHmiTimesDay[7].shift[3].break[0..4].endCircuitTime := TOD#00:00:00;
   statHmiTimesDay[0].shift[0].break[0..4].end := TOD#00:00:00;
   statHmiTimesDay[0].shift[1].break[0..4].end := TOD#00:00:00;
   statHmiTimesDay[0].shift[2].break[0..4].end := TOD#00:00:00;
   statHmiTimesDay[0].shift[3].break[0..4].end := TOD#00:00:00;
   statHmiTimesDay[1].shift[0].break[0..4].end := TOD#00:00:00;
   statHmiTimesDay[1].shift[1].break[0..4].end := TOD#00:00:00;
   statHmiTimesDay[1].shift[2].break[0..4].end := TOD#00:00:00;
   statHmiTimesDay[1].shift[3].break[0..4].end := TOD#00:00:00;
   statHmiTimesDay[2].shift[0].break[0..4].end := TOD#00:00:00;
   statHmiTimesDay[2].shift[1].break[0..4].end := TOD#00:00:00;
   statHmiTimesDay[2].shift[2].break[0..4].end := TOD#00:00:00;
   statHmiTimesDay[2].shift[3].break[0..4].end := TOD#00:00:00;
   statHmiTimesDay[3].shift[0].break[0..4].end := TOD#00:00:00;
   statHmiTimesDay[3].shift[1].break[0..4].end := TOD#00:00:00;
   statHmiTimesDay[3].shift[2].break[0..4].end := TOD#00:00:00;
   statHmiTimesDay[3].shift[3].break[0..4].end := TOD#00:00:00;
   statHmiTimesDay[4].shift[0].break[0..4].end := TOD#00:00:00;
   statHmiTimesDay[4].shift[1].break[0..4].end := TOD#00:00:00;
   statHmiTimesDay[4].shift[2].break[0..4].end := TOD#00:00:00;
   statHmiTimesDay[4].shift[3].break[0..4].end := TOD#00:00:00;
   statHmiTimesDay[5].shift[0].break[0..4].end := TOD#00:00:00;
   statHmiTimesDay[5].shift[1].break[0..4].end := TOD#00:00:00;
   statHmiTimesDay[5].shift[2].break[0..4].end := TOD#00:00:00;
   statHmiTimesDay[5].shift[3].break[0..4].end := TOD#00:00:00;
   statHmiTimesDay[6].shift[0].break[0..4].end := TOD#00:00:00;
   statHmiTimesDay[6].shift[1].break[0..4].end := TOD#00:00:00;
   statHmiTimesDay[6].shift[2].break[0..4].end := TOD#00:00:00;
   statHmiTimesDay[6].shift[3].break[0..4].end := TOD#00:00:00;
   statHmiTimesDay[7].shift[0].break[0..4].end := TOD#00:00:00;
   statHmiTimesDay[7].shift[1].break[0..4].end := TOD#00:00:00;
   statHmiTimesDay[7].shift[2].break[0..4].end := TOD#00:00:00;
   statHmiTimesDay[7].shift[3].break[0..4].end := TOD#00:00:00;
   statHmiTimesDay[0].shift[0..3].end := TOD#00:00:00;
   statHmiTimesDay[1].shift[0..3].end := TOD#00:00:00;
   statHmiTimesDay[2].shift[0..3].end := TOD#00:00:00;
   statHmiTimesDay[3].shift[0..3].end := TOD#00:00:00;
   statHmiTimesDay[4].shift[0..3].end := TOD#00:00:00;
   statHmiTimesDay[5].shift[0..3].end := TOD#00:00:00;
   statHmiTimesDay[6].shift[0..3].end := TOD#00:00:00;
   statHmiTimesDay[7].shift[0..3].end := TOD#00:00:00;
   statHmiTimesDay[0].shift[0..3].startCircuitTime := TOD#00:00:00;
   statHmiTimesDay[1].shift[0..3].startCircuitTime := TOD#00:00:00;
   statHmiTimesDay[2].shift[0..3].startCircuitTime := TOD#00:00:00;
   statHmiTimesDay[3].shift[0..3].startCircuitTime := TOD#00:00:00;
   statHmiTimesDay[4].shift[0..3].startCircuitTime := TOD#00:00:00;
   statHmiTimesDay[5].shift[0..3].startCircuitTime := TOD#00:00:00;
   statHmiTimesDay[6].shift[0..3].startCircuitTime := TOD#00:00:00;
   statHmiTimesDay[7].shift[0..3].startCircuitTime := TOD#00:00:00;
   statHmiSignalsDay[0].shift[0..3].shiftConfig := FALSE;
   statHmiSignalsDay[1].shift[0..3].shiftConfig := FALSE;
   statHmiSignalsDay[2].shift[0..3].shiftConfig := FALSE;
   statHmiSignalsDay[3].shift[0..3].shiftConfig := FALSE;
   statHmiSignalsDay[4].shift[0..3].shiftConfig := FALSE;
   statHmiSignalsDay[5].shift[0..3].shiftConfig := FALSE;
   statHmiSignalsDay[6].shift[0..3].shiftConfig := FALSE;
   statHmiSignalsDay[7].shift[0..3].shiftConfig := FALSE;
   statHmiSignalsDay[0].shift[0..3].shiftActive := FALSE;
   statHmiSignalsDay[1].shift[0..3].shiftActive := FALSE;
   statHmiSignalsDay[2].shift[0..3].shiftActive := FALSE;
   statHmiSignalsDay[3].shift[0..3].shiftActive := FALSE;
   statHmiSignalsDay[4].shift[0..3].shiftActive := FALSE;
   statHmiSignalsDay[5].shift[0..3].shiftActive := FALSE;
   statHmiSignalsDay[6].shift[0..3].shiftActive := FALSE;
   statHmiSignalsDay[7].shift[0..3].shiftActive := FALSE;
   statHmiSignalsDay[0].shift[0..3].shiftEndCirTimeConfig := FALSE;
   statHmiSignalsDay[1].shift[0..3].shiftEndCirTimeConfig := FALSE;
   statHmiSignalsDay[2].shift[0..3].shiftEndCirTimeConfig := FALSE;
   statHmiSignalsDay[3].shift[0..3].shiftEndCirTimeConfig := FALSE;
   statHmiSignalsDay[4].shift[0..3].shiftEndCirTimeConfig := FALSE;
   statHmiSignalsDay[5].shift[0..3].shiftEndCirTimeConfig := FALSE;
   statHmiSignalsDay[6].shift[0..3].shiftEndCirTimeConfig := FALSE;
   statHmiSignalsDay[7].shift[0..3].shiftEndCirTimeConfig := FALSE;
   statHmiSignalsDay[0].shift[0..3].shiftStartCirTimeConfig := FALSE;
   statHmiSignalsDay[1].shift[0..3].shiftStartCirTimeConfig := FALSE;
   statHmiSignalsDay[2].shift[0..3].shiftStartCirTimeConfig := FALSE;
   statHmiSignalsDay[3].shift[0..3].shiftStartCirTimeConfig := FALSE;
   statHmiSignalsDay[4].shift[0..3].shiftStartCirTimeConfig := FALSE;
   statHmiSignalsDay[5].shift[0..3].shiftStartCirTimeConfig := FALSE;
   statHmiSignalsDay[6].shift[0..3].shiftStartCirTimeConfig := FALSE;
   statHmiSignalsDay[7].shift[0..3].shiftStartCirTimeConfig := FALSE;
   statHmiSignalsDay[0].shift[0..3].shiftEndCirTimeActive := FALSE;
   statHmiSignalsDay[1].shift[0..3].shiftEndCirTimeActive := FALSE;
   statHmiSignalsDay[2].shift[0..3].shiftEndCirTimeActive := FALSE;
   statHmiSignalsDay[3].shift[0..3].shiftEndCirTimeActive := FALSE;
   statHmiSignalsDay[4].shift[0..3].shiftEndCirTimeActive := FALSE;
   statHmiSignalsDay[5].shift[0..3].shiftEndCirTimeActive := FALSE;
   statHmiSignalsDay[6].shift[0..3].shiftEndCirTimeActive := FALSE;
   statHmiSignalsDay[7].shift[0..3].shiftEndCirTimeActive := FALSE;
   statHmiSignalsDay[0].shift[0..3].shiftStartCirTimeActive := FALSE;
   statHmiSignalsDay[1].shift[0..3].shiftStartCirTimeActive := FALSE;
   statHmiSignalsDay[2].shift[0..3].shiftStartCirTimeActive := FALSE;
   statHmiSignalsDay[3].shift[0..3].shiftStartCirTimeActive := FALSE;
   statHmiSignalsDay[4].shift[0..3].shiftStartCirTimeActive := FALSE;
   statHmiSignalsDay[5].shift[0..3].shiftStartCirTimeActive := FALSE;
   statHmiSignalsDay[6].shift[0..3].shiftStartCirTimeActive := FALSE;
   statHmiSignalsDay[7].shift[0..3].shiftStartCirTimeActive := FALSE;
   statHmiSignalsDay[0].shift[0..3].shiftSignalsHmi := 16#00;
   statHmiSignalsDay[1].shift[0..3].shiftSignalsHmi := 16#00;
   statHmiSignalsDay[2].shift[0..3].shiftSignalsHmi := 16#00;
   statHmiSignalsDay[3].shift[0..3].shiftSignalsHmi := 16#00;
   statHmiSignalsDay[4].shift[0..3].shiftSignalsHmi := 16#00;
   statHmiSignalsDay[5].shift[0..3].shiftSignalsHmi := 16#00;
   statHmiSignalsDay[6].shift[0..3].shiftSignalsHmi := 16#00;
   statHmiSignalsDay[7].shift[0..3].shiftSignalsHmi := 16#00;
   statHmiSignalsDay[0].shift[0].break[0..4].config := FALSE;
   statHmiSignalsDay[0].shift[1].break[0..4].config := FALSE;
   statHmiSignalsDay[0].shift[2].break[0..4].config := FALSE;
   statHmiSignalsDay[0].shift[3].break[0..4].config := FALSE;
   statHmiSignalsDay[1].shift[0].break[0..4].config := FALSE;
   statHmiSignalsDay[1].shift[1].break[0..4].config := FALSE;
   statHmiSignalsDay[1].shift[2].break[0..4].config := FALSE;
   statHmiSignalsDay[1].shift[3].break[0..4].config := FALSE;
   statHmiSignalsDay[2].shift[0].break[0..4].config := FALSE;
   statHmiSignalsDay[2].shift[1].break[0..4].config := FALSE;
   statHmiSignalsDay[2].shift[2].break[0..4].config := FALSE;
   statHmiSignalsDay[2].shift[3].break[0..4].config := FALSE;
   statHmiSignalsDay[3].shift[0].break[0..4].config := FALSE;
   statHmiSignalsDay[3].shift[1].break[0..4].config := FALSE;
   statHmiSignalsDay[3].shift[2].break[0..4].config := FALSE;
   statHmiSignalsDay[3].shift[3].break[0..4].config := FALSE;
   statHmiSignalsDay[4].shift[0].break[0..4].config := FALSE;
   statHmiSignalsDay[4].shift[1].break[0..4].config := FALSE;
   statHmiSignalsDay[4].shift[2].break[0..4].config := FALSE;
   statHmiSignalsDay[4].shift[3].break[0..4].config := FALSE;
   statHmiSignalsDay[5].shift[0].break[0..4].config := FALSE;
   statHmiSignalsDay[5].shift[1].break[0..4].config := FALSE;
   statHmiSignalsDay[5].shift[2].break[0..4].config := FALSE;
   statHmiSignalsDay[5].shift[3].break[0..4].config := FALSE;
   statHmiSignalsDay[6].shift[0].break[0..4].config := FALSE;
   statHmiSignalsDay[6].shift[1].break[0..4].config := FALSE;
   statHmiSignalsDay[6].shift[2].break[0..4].config := FALSE;
   statHmiSignalsDay[6].shift[3].break[0..4].config := FALSE;
   statHmiSignalsDay[7].shift[0].break[0..4].config := FALSE;
   statHmiSignalsDay[7].shift[1].break[0..4].config := FALSE;
   statHmiSignalsDay[7].shift[2].break[0..4].config := FALSE;
   statHmiSignalsDay[7].shift[3].break[0..4].config := FALSE;
   statHmiSignalsDay[0].shift[0].break[0..4].active := FALSE;
   statHmiSignalsDay[0].shift[1].break[0..4].active := FALSE;
   statHmiSignalsDay[0].shift[2].break[0..4].active := FALSE;
   statHmiSignalsDay[0].shift[3].break[0..4].active := FALSE;
   statHmiSignalsDay[1].shift[0].break[0..4].active := FALSE;
   statHmiSignalsDay[1].shift[1].break[0..4].active := FALSE;
   statHmiSignalsDay[1].shift[2].break[0..4].active := FALSE;
   statHmiSignalsDay[1].shift[3].break[0..4].active := FALSE;
   statHmiSignalsDay[2].shift[0].break[0..4].active := FALSE;
   statHmiSignalsDay[2].shift[1].break[0..4].active := FALSE;
   statHmiSignalsDay[2].shift[2].break[0..4].active := FALSE;
   statHmiSignalsDay[2].shift[3].break[0..4].active := FALSE;
   statHmiSignalsDay[3].shift[0].break[0..4].active := FALSE;
   statHmiSignalsDay[3].shift[1].break[0..4].active := FALSE;
   statHmiSignalsDay[3].shift[2].break[0..4].active := FALSE;
   statHmiSignalsDay[3].shift[3].break[0..4].active := FALSE;
   statHmiSignalsDay[4].shift[0].break[0..4].active := FALSE;
   statHmiSignalsDay[4].shift[1].break[0..4].active := FALSE;
   statHmiSignalsDay[4].shift[2].break[0..4].active := FALSE;
   statHmiSignalsDay[4].shift[3].break[0..4].active := FALSE;
   statHmiSignalsDay[5].shift[0].break[0..4].active := FALSE;
   statHmiSignalsDay[5].shift[1].break[0..4].active := FALSE;
   statHmiSignalsDay[5].shift[2].break[0..4].active := FALSE;
   statHmiSignalsDay[5].shift[3].break[0..4].active := FALSE;
   statHmiSignalsDay[6].shift[0].break[0..4].active := FALSE;
   statHmiSignalsDay[6].shift[1].break[0..4].active := FALSE;
   statHmiSignalsDay[6].shift[2].break[0..4].active := FALSE;
   statHmiSignalsDay[6].shift[3].break[0..4].active := FALSE;
   statHmiSignalsDay[7].shift[0].break[0..4].active := FALSE;
   statHmiSignalsDay[7].shift[1].break[0..4].active := FALSE;
   statHmiSignalsDay[7].shift[2].break[0..4].active := FALSE;
   statHmiSignalsDay[7].shift[3].break[0..4].active := FALSE;
   statHmiSignalsDay[0].shift[0].break[0..4].circuitTimeConfig := FALSE;
   statHmiSignalsDay[0].shift[1].break[0..4].circuitTimeConfig := FALSE;
   statHmiSignalsDay[0].shift[2].break[0..4].circuitTimeConfig := FALSE;
   statHmiSignalsDay[0].shift[3].break[0..4].circuitTimeConfig := FALSE;
   statHmiSignalsDay[1].shift[0].break[0..4].circuitTimeConfig := FALSE;
   statHmiSignalsDay[1].shift[1].break[0..4].circuitTimeConfig := FALSE;
   statHmiSignalsDay[1].shift[2].break[0..4].circuitTimeConfig := FALSE;
   statHmiSignalsDay[1].shift[3].break[0..4].circuitTimeConfig := FALSE;
   statHmiSignalsDay[2].shift[0].break[0..4].circuitTimeConfig := FALSE;
   statHmiSignalsDay[2].shift[1].break[0..4].circuitTimeConfig := FALSE;
   statHmiSignalsDay[2].shift[2].break[0..4].circuitTimeConfig := FALSE;
   statHmiSignalsDay[2].shift[3].break[0..4].circuitTimeConfig := FALSE;
   statHmiSignalsDay[3].shift[0].break[0..4].circuitTimeConfig := FALSE;
   statHmiSignalsDay[3].shift[1].break[0..4].circuitTimeConfig := FALSE;
   statHmiSignalsDay[3].shift[2].break[0..4].circuitTimeConfig := FALSE;
   statHmiSignalsDay[3].shift[3].break[0..4].circuitTimeConfig := FALSE;
   statHmiSignalsDay[4].shift[0].break[0..4].circuitTimeConfig := FALSE;
   statHmiSignalsDay[4].shift[1].break[0..4].circuitTimeConfig := FALSE;
   statHmiSignalsDay[4].shift[2].break[0..4].circuitTimeConfig := FALSE;
   statHmiSignalsDay[4].shift[3].break[0..4].circuitTimeConfig := FALSE;
   statHmiSignalsDay[5].shift[0].break[0..4].circuitTimeConfig := FALSE;
   statHmiSignalsDay[5].shift[1].break[0..4].circuitTimeConfig := FALSE;
   statHmiSignalsDay[5].shift[2].break[0..4].circuitTimeConfig := FALSE;
   statHmiSignalsDay[5].shift[3].break[0..4].circuitTimeConfig := FALSE;
   statHmiSignalsDay[6].shift[0].break[0..4].circuitTimeConfig := FALSE;
   statHmiSignalsDay[6].shift[1].break[0..4].circuitTimeConfig := FALSE;
   statHmiSignalsDay[6].shift[2].break[0..4].circuitTimeConfig := FALSE;
   statHmiSignalsDay[6].shift[3].break[0..4].circuitTimeConfig := FALSE;
   statHmiSignalsDay[7].shift[0].break[0..4].circuitTimeConfig := FALSE;
   statHmiSignalsDay[7].shift[1].break[0..4].circuitTimeConfig := FALSE;
   statHmiSignalsDay[7].shift[2].break[0..4].circuitTimeConfig := FALSE;
   statHmiSignalsDay[7].shift[3].break[0..4].circuitTimeConfig := FALSE;
   statHmiSignalsDay[0].shift[0].break[0..4].circuitTimeActive := FALSE;
   statHmiSignalsDay[0].shift[1].break[0..4].circuitTimeActive := FALSE;
   statHmiSignalsDay[0].shift[2].break[0..4].circuitTimeActive := FALSE;
   statHmiSignalsDay[0].shift[3].break[0..4].circuitTimeActive := FALSE;
   statHmiSignalsDay[1].shift[0].break[0..4].circuitTimeActive := FALSE;
   statHmiSignalsDay[1].shift[1].break[0..4].circuitTimeActive := FALSE;
   statHmiSignalsDay[1].shift[2].break[0..4].circuitTimeActive := FALSE;
   statHmiSignalsDay[1].shift[3].break[0..4].circuitTimeActive := FALSE;
   statHmiSignalsDay[2].shift[0].break[0..4].circuitTimeActive := FALSE;
   statHmiSignalsDay[2].shift[1].break[0..4].circuitTimeActive := FALSE;
   statHmiSignalsDay[2].shift[2].break[0..4].circuitTimeActive := FALSE;
   statHmiSignalsDay[2].shift[3].break[0..4].circuitTimeActive := FALSE;
   statHmiSignalsDay[3].shift[0].break[0..4].circuitTimeActive := FALSE;
   statHmiSignalsDay[3].shift[1].break[0..4].circuitTimeActive := FALSE;
   statHmiSignalsDay[3].shift[2].break[0..4].circuitTimeActive := FALSE;
   statHmiSignalsDay[3].shift[3].break[0..4].circuitTimeActive := FALSE;
   statHmiSignalsDay[4].shift[0].break[0..4].circuitTimeActive := FALSE;
   statHmiSignalsDay[4].shift[1].break[0..4].circuitTimeActive := FALSE;
   statHmiSignalsDay[4].shift[2].break[0..4].circuitTimeActive := FALSE;
   statHmiSignalsDay[4].shift[3].break[0..4].circuitTimeActive := FALSE;
   statHmiSignalsDay[5].shift[0].break[0..4].circuitTimeActive := FALSE;
   statHmiSignalsDay[5].shift[1].break[0..4].circuitTimeActive := FALSE;
   statHmiSignalsDay[5].shift[2].break[0..4].circuitTimeActive := FALSE;
   statHmiSignalsDay[5].shift[3].break[0..4].circuitTimeActive := FALSE;
   statHmiSignalsDay[6].shift[0].break[0..4].circuitTimeActive := FALSE;
   statHmiSignalsDay[6].shift[1].break[0..4].circuitTimeActive := FALSE;
   statHmiSignalsDay[6].shift[2].break[0..4].circuitTimeActive := FALSE;
   statHmiSignalsDay[6].shift[3].break[0..4].circuitTimeActive := FALSE;
   statHmiSignalsDay[7].shift[0].break[0..4].circuitTimeActive := FALSE;
   statHmiSignalsDay[7].shift[1].break[0..4].circuitTimeActive := FALSE;
   statHmiSignalsDay[7].shift[2].break[0..4].circuitTimeActive := FALSE;
   statHmiSignalsDay[7].shift[3].break[0..4].circuitTimeActive := FALSE;
   statHmiSignalsDay[0].shift[0..3].breakSignalsHmi := 16#0000;
   statHmiSignalsDay[1].shift[0..3].breakSignalsHmi := 16#0000;
   statHmiSignalsDay[2].shift[0..3].breakSignalsHmi := 16#0000;
   statHmiSignalsDay[3].shift[0..3].breakSignalsHmi := 16#0000;
   statHmiSignalsDay[4].shift[0..3].breakSignalsHmi := 16#0000;
   statHmiSignalsDay[5].shift[0..3].breakSignalsHmi := 16#0000;
   statHmiSignalsDay[6].shift[0..3].breakSignalsHmi := 16#0000;
   statHmiSignalsDay[7].shift[0..3].breakSignalsHmi := 16#0000;
   statHmiSignalsDay[0..7].shiftsPerDay := 0;
   statSummaryHmi.earlyShiftActive := FALSE;
   statSummaryHmi.lateShiftActive := FALSE;
   statSummaryHmi.nightShiftActive := FALSE;
   statSummaryHmi.breakInShiftActive := FALSE;
   statSummaryHmi.breakBetweenShiftAct := FALSE;
   statSummaryHmi.breakActive := FALSE;
   statSummaryHmi.circuitTimeInShiftAct := FALSE;
   statSummaryHmi.circuitTimeBetwShiftAct := FALSE;
   statSummaryHmi.circuitTimeActive := FALSE;
   statSummaryHmi.noOfWorkdays := 0;
   statSummaryHmi.workdays[0..7] := FALSE;
   statZeroDay.shift[0..3].endCircuitTime := TOD#00:00:00;
   statZeroDay.shift[0..3].start := TOD#00:00:00;
   statZeroDay.shift[0].break[0..4].start := TOD#00:00:00;
   statZeroDay.shift[1].break[0..4].start := TOD#00:00:00;
   statZeroDay.shift[2].break[0..4].start := TOD#00:00:00;
   statZeroDay.shift[3].break[0..4].start := TOD#00:00:00;
   statZeroDay.shift[0].break[0..4].startCircuitTime := TOD#00:00:00;
   statZeroDay.shift[1].break[0..4].startCircuitTime := TOD#00:00:00;
   statZeroDay.shift[2].break[0..4].startCircuitTime := TOD#00:00:00;
   statZeroDay.shift[3].break[0..4].startCircuitTime := TOD#00:00:00;
   statZeroDay.shift[0].break[0..4].endCircuitTime := TOD#00:00:00;
   statZeroDay.shift[1].break[0..4].endCircuitTime := TOD#00:00:00;
   statZeroDay.shift[2].break[0..4].endCircuitTime := TOD#00:00:00;
   statZeroDay.shift[3].break[0..4].endCircuitTime := TOD#00:00:00;
   statZeroDay.shift[0].break[0..4].end := TOD#00:00:00;
   statZeroDay.shift[1].break[0..4].end := TOD#00:00:00;
   statZeroDay.shift[2].break[0..4].end := TOD#00:00:00;
   statZeroDay.shift[3].break[0..4].end := TOD#00:00:00;
   statZeroDay.shift[0..3].end := TOD#00:00:00;
   statZeroDay.shift[0..3].startCircuitTime := TOD#00:00:00;
   statCheckCircuitTime.startTime := TOD#00:00:00;
   statCheckCircuitTime.fromDay := 1;
   statCheckCircuitTime.fromShift := 1;
   statCheckCircuitTime.endTime := TOD#00:00:00;
   statCheckCircuitTime.toDay := 1;
   statCheckCircuitTime.toShift := 1;
   statRisEdge.earlyShiftActive := FALSE;
   statRisEdge.lateShiftActive := FALSE;
   statRisEdge.nightShiftActive := FALSE;
   statRisEdge.breakInShiftActive := FALSE;
   statRisEdge.breakBetweenShiftAct := FALSE;
   statRisEdge.breakActive := FALSE;
   statRisEdge.circuitTimeInShiftAct := FALSE;
   statRisEdge.circuitTimeBetwShiftAct := FALSE;
   statRisEdge.circuitTimeActive := FALSE;
   statRisEdge.noOfWorkdays := 0;
   statRisEdge.workdays[0..7] := FALSE;
   statPosPulse.earlyShiftActive := FALSE;
   statPosPulse.lateShiftActive := FALSE;
   statPosPulse.nightShiftActive := FALSE;
   statPosPulse.breakInShiftActive := FALSE;
   statPosPulse.breakBetweenShiftAct := FALSE;
   statPosPulse.breakActive := FALSE;
   statPosPulse.circuitTimeInShiftAct := FALSE;
   statPosPulse.circuitTimeBetwShiftAct := FALSE;
   statPosPulse.circuitTimeActive := FALSE;
   statPosPulse.noOfWorkdays := 0;
   statPosPulse.workdays[0..7] := FALSE;
   statFalEdge.earlyShiftActive := FALSE;
   statFalEdge.lateShiftActive := FALSE;
   statFalEdge.nightShiftActive := FALSE;
   statFalEdge.breakInShiftActive := FALSE;
   statFalEdge.breakBetweenShiftAct := FALSE;
   statFalEdge.breakActive := FALSE;
   statFalEdge.circuitTimeInShiftAct := FALSE;
   statFalEdge.circuitTimeBetwShiftAct := FALSE;
   statFalEdge.circuitTimeActive := FALSE;
   statFalEdge.noOfWorkdays := 0;
   statFalEdge.workdays[0..7] := FALSE;
   statNegPulse.earlyShiftActive := FALSE;
   statNegPulse.lateShiftActive := FALSE;
   statNegPulse.nightShiftActive := FALSE;
   statNegPulse.breakInShiftActive := FALSE;
   statNegPulse.breakBetweenShiftAct := FALSE;
   statNegPulse.breakActive := FALSE;
   statNegPulse.circuitTimeInShiftAct := FALSE;
   statNegPulse.circuitTimeBetwShiftAct := FALSE;
   statNegPulse.circuitTimeActive := FALSE;
   statNegPulse.noOfWorkdays := 0;
   statNegPulse.workdays[0..7] := FALSE;
   statTimesAndCircuit.endCircuitTime := TOD#00:00:00;
   statTimesAndCircuit.start := TOD#00:00:00;
   statTimesAndCircuit.break[0..4].start := TOD#00:00:00;
   statTimesAndCircuit.break[0..4].startCircuitTime := TOD#00:00:00;
   statTimesAndCircuit.break[0..4].endCircuitTime := TOD#00:00:00;
   statTimesAndCircuit.break[0..4].end := TOD#00:00:00;
   statTimesAndCircuit.end := TOD#00:00:00;
   statTimesAndCircuit.startCircuitTime := TOD#00:00:00;
   statOnlyTimes.start := TOD#00:00:00;
   statOnlyTimes.break[0..4].start := TOD#00:00:00;
   statOnlyTimes.break[0..4].startCircuitTime := TOD#00:00:00;
   statOnlyTimes.break[0..4].endCircuitTime := TOD#00:00:00;
   statOnlyTimes.break[0..4].end := TOD#00:00:00;
   statOnlyTimes.end := TOD#00:00:00;
END_DATA_BLOCK

DATA_BLOCK "EeMonitor"   // DB61
TITLE = EeMonitor
AUTHOR : SICAR
FAMILY : DB
// Globale EEM Informationen / Global EEM Information
// stored: InstanceOfName LSicar_typeEemDataHmi, InstanceOfType UDT
"LSicar_typeEemDataHmi"
   // VAR
   //    measurePointIndex : USInt := 0;
   //    measConfiguration { ExternalWritable := 'False'} : EnS_EEm_typeMeasConfig;
   //    measOperationHmi { ExternalWritable := 'False'} : EnS_EEm_typeMeasOperation;
   //    work { ExternalWritable := 'False'} : "LSicar_typeEnMeterWorkHmi";
   // END_VAR
BEGIN
   measConfiguration."name" := 'AIEnergyMeter480VACST_EM01';
   measConfiguration.nameShort := 'EM01';
   measConfiguration.media := 'electrical';
   measConfiguration.unitCounterNumber := 1;
   measConfiguration.unitCounterText := 'Wh';
   measConfiguration.unitActValueNumber := 0;
   measConfiguration.unitActValueText := 'W';
   measConfiguration.inputType := 1;
   measConfiguration.type1Counter.overflowCntValue := 1000000.0;
   measConfiguration.type1Counter.normFactor := 1.0;
   measConfiguration.type2ActValue.rawLow := 0.0;
   measConfiguration.type2ActValue.rawHigh := 100.0;
   measConfiguration.type2ActValue.outLow := 0.0;
   measConfiguration.type2ActValue.outHigh := 100.0;
   measOperationHmi.in.counterValue := 277.384918212891;
   measOperationHmi.in.actValue := 0.0;
   measOperationHmi.out.avgValue[0..8] := 0.0;
   measOperationHmi.out.refValue[0..8] := 0.0;
   measOperationHmi.out.differencePercent[0..8] := 0.0;
   measOperationHmi.out.energyCounter[0] := 4.5557861328125;
   measOperationHmi.out.energyCounter[1..8] := 0.0;
   measOperationHmi.out.energyCounterTotal := 4.5557861328125;
   measOperationHmi.out.error := FALSE;
   measOperationHmi.out.energyPerItem := 0.0;
   measOperationHmi.stat.counterLast := 277.473693847656;
   measOperationHmi.stat.counterDifference := 277.384918212891;
   measOperationHmi.stat.startEnergyValue[0..8] := 0.0;
   measOperationHmi.stat.energyCounterIntermediate := 0.0;
   measOperationHmi.stat.energyEnPiCalc[0] := 4.555786;
   measOperationHmi.stat.energyEnPiCalc[1..8] := 0.0;
   work.cycleCounterAvgCalcTod := TOD#00:00:00;
   work.cycleCounterAvgCalcDtl := DTL#1970-01-01-00:00:00;
   work.timePeriodAvgValTod := TOD#00:00:00;
   work.timePeriodAvgValDtl := DTL#1970-01-01-00:00:00;
   work.timePeriodAvgRefTod := TOD#00:00:00;
   work.timePeriodAvgRefDtl := DTL#1970-01-01-00:00:00;
   work.startTimeAvgValLocTime := DTL#1970-01-01-00:00:00;
   work.startTimeAvgRefLocTime := DTL#1970-01-01-00:00:00;
   work.numberOfRecords := 209;
END_DATA_BLOCK

DATA_BLOCK "EeMonitorData"   // DB108
TITLE = EeMonitorData
AUTHOR : SICAR
FAMILY : DB
// Energy efficency monitor Daten / Energy efficency monitor data
// stored: InstanceOfName LSicar_typeEemData, InstanceOfType UDT
"LSicar_typeEemData"
   // VAR
   //    machineConfiguration : EnS_EEm_typeConfig;
   //    machineOperation : EnS_EEm_typeOperation;
   //    measConfiguration : Array[0..9] of EnS_EEm_typeMeasConfig;
   //    measOperation : Array[0..9] of EnS_EEm_typeMeasOperation;
   //    internalData : "LSicar_typeEemDataInternal";
   //    calcError : Bool := FALSE;
   //    calcStatus : Word := 16#740B;
   //    calcRetVal : Int := 0;
   //    reportCreateCsv : Bool := FALSE;
   //    reportStatus : Word := 16#0000;
   //    reportNameCsv : String[80] := '';
   // END_VAR
BEGIN
   machineConfiguration."name" := 'Default_Machine_Demo';
   machineConfiguration."type" := 'Default_Type_Demo';
   machineConfiguration.serialNumber := 'Default_Serial_Number_Demo';
   machineConfiguration.manufacturer := 'Default_Manufacturer_Demo';
   machineConfiguration.licenseKey := 'Demo_Demo_Demo_Demo!';
   machineConfiguration.pieceOverflowCntValue := 10000.0;
   machineConfiguration.eStateName[0] := 'Undefined';
   machineConfiguration.eStateName[1] := 'Auto';
   machineConfiguration.eStateName[2] := 'Auto Preselect';
   machineConfiguration.eStateName[3] := 'Manual';
   machineConfiguration.eStateName[4] := 'Idle';
   machineConfiguration.eStateName[5] := 'Fault';
   machineConfiguration.eStateName[6..8] := '-Not used-';
   machineConfiguration.additionalInfoDescription[0] := 'additional Info1';
   machineConfiguration.additionalInfoDescription[1] := 'additional Info2';
   machineConfiguration.additionalInfoDescription[2] := 'additional Info3';
   machineConfiguration.additionalInfoDescription[3] := 'additional Info4';
   machineOperation.pieceCounter := 0.0;
   machineOperation.additionalInformation[0] := 'AddInfo 1';
   machineOperation.additionalInformation[1] := 'AddInfo 2';
   machineOperation.additionalInformation[2] := 'AddInfo 3';
   machineOperation.additionalInformation[3] := 'AddInfo 4';
   machineOperation.eState := 0;
   machineOperation.maskEnPI := 16#0002;
   machineOperation.triggerRecalcOutput := FALSE;
   machineOperation.resetMeasErrors := FALSE;
   machineOperation.globalResetEnergyCounter := FALSE;
   machineOperation.globalResetAvgValues := FALSE;
   machineOperation.globalResetEnergyPerItem := FALSE;
   machineOperation.startAvgCalcPeriod := FALSE;
   machineOperation.stopAvgCalcPeriod := FALSE;
   machineOperation.setAvgCalcRef := FALSE;
   machineOperation.stat.arraysOk := TRUE;
   machineOperation.stat.avgCalcAct := FALSE;
   machineOperation.stat.triggerRecalcOld := FALSE;
   machineOperation.stat.startAvgCalcOld := FALSE;
   machineOperation.stat.stopAvgCalcOld := FALSE;
   machineOperation.stat.referenceAvgCalcSave := FALSE;
   machineOperation.stat.outputValuesRelease := TRUE;
   machineOperation.stat.maskEnpiOld := 16#0002;
   machineOperation.stat.machineEStateOld := 0;
   machineOperation.stat.upBoundMeasConfiguration := 9;
   machineOperation.stat.upBoundMeasOperation := 9;
   machineOperation.stat.lowBoundMeasConfiguration := 0;
   machineOperation.stat.lowBoundMeasOperation := 0;
   machineOperation.stat.pieceCntOld := 0.0;
   machineOperation.stat.pieceCntEnpiCalc := 0.0;
   machineOperation.stat.cycleCounterAvgCalc := 0;
   machineOperation.stat.cycleCounterEstates[0..8] := 0;
   machineOperation.stat.startTimeAvgVal := DTL#1970-01-01-00:00:00;
   machineOperation.stat.timePeriodAvgVal := T#0MS;
   machineOperation.stat.timeZoneValues := T#0MS;
   machineOperation.stat.startTimeAvgRef := DTL#1970-01-01-00:00:00;
   machineOperation.stat.timePeriodAvgRef := T#0MS;
   machineOperation.stat.timeZoneRef := T#0MS;
   machineOperation.stat.systemInformation[0] := 16#07;
   machineOperation.stat.systemInformation[1] := 16#EA;
   machineOperation.stat.systemInformation[2] := 16#01;
   machineOperation.stat.systemInformation[3] := 16#06;
   machineOperation.stat.systemInformation[4] := 16#03;
   machineOperation.stat.systemInformation[5] := 16#05;
   machineOperation.stat.systemInformation[6] := 16#09;
   machineOperation.stat.systemInformation[7] := 16#2B;
   machineOperation.stat.systemInformation[8] := 16#03;
   machineOperation.stat.systemInformation[9] := 16#CC;
   machineOperation.stat.systemInformation[10] := 16#19;
   machineOperation.stat.systemInformation[11] := 16#C5;
   measConfiguration[0]."name" := 'AIEnergyMeter480VACST_EM01';
   measConfiguration[1]."name" := 'AIEnergyMeter480VACST_EM02';
   measConfiguration[2]."name" := 'PAC Electrical Infeed';
   measConfiguration[3..9]."name" := 'MeasPointXX';
   measConfiguration[0].nameShort := 'EM01';
   measConfiguration[1].nameShort := 'EM02';
   measConfiguration[2].nameShort := 'P01';
   measConfiguration[3..9].nameShort := 'XX01';
   measConfiguration[0..9].media := 'electrical';
   measConfiguration[0..9].unitCounterNumber := 1;
   measConfiguration[0..9].unitCounterText := 'Wh';
   measConfiguration[0..9].unitActValueNumber := 0;
   measConfiguration[0..9].unitActValueText := 'W';
   measConfiguration[0..9].inputType := 1;
   measConfiguration[0..9].type1Counter.overflowCntValue := 1000000.0;
   measConfiguration[0..9].type1Counter.normFactor := 1.0;
   measConfiguration[0..9].type2ActValue.rawLow := 0.0;
   measConfiguration[0..9].type2ActValue.rawHigh := 100.0;
   measConfiguration[0..9].type2ActValue.outLow := 0.0;
   measConfiguration[0..9].type2ActValue.outHigh := 100.0;
   measOperation[0].in.counterValue := 277.384918212891;
   measOperation[1..9].in.counterValue := 0.0;
   measOperation[0..9].in.actValue := 0.0;
   measOperation[0].out.avgValue[0..8] := 0.0;
   measOperation[1].out.avgValue[0..8] := 0.0;
   measOperation[2].out.avgValue[0..8] := 0.0;
   measOperation[3].out.avgValue[0..8] := 0.0;
   measOperation[4].out.avgValue[0..8] := 0.0;
   measOperation[5].out.avgValue[0..8] := 0.0;
   measOperation[6].out.avgValue[0..8] := 0.0;
   measOperation[7].out.avgValue[0..8] := 0.0;
   measOperation[8].out.avgValue[0..8] := 0.0;
   measOperation[9].out.avgValue[0..8] := 0.0;
   measOperation[0].out.refValue[0..8] := 0.0;
   measOperation[1].out.refValue[0..8] := 0.0;
   measOperation[2].out.refValue[0..8] := 0.0;
   measOperation[3].out.refValue[0..8] := 0.0;
   measOperation[4].out.refValue[0..8] := 0.0;
   measOperation[5].out.refValue[0..8] := 0.0;
   measOperation[6].out.refValue[0..8] := 0.0;
   measOperation[7].out.refValue[0..8] := 0.0;
   measOperation[8].out.refValue[0..8] := 0.0;
   measOperation[9].out.refValue[0..8] := 0.0;
   measOperation[0].out.differencePercent[0..8] := 0.0;
   measOperation[1].out.differencePercent[0..8] := 0.0;
   measOperation[2].out.differencePercent[0..8] := 0.0;
   measOperation[3].out.differencePercent[0..8] := 0.0;
   measOperation[4].out.differencePercent[0..8] := 0.0;
   measOperation[5].out.differencePercent[0..8] := 0.0;
   measOperation[6].out.differencePercent[0..8] := 0.0;
   measOperation[7].out.differencePercent[0..8] := 0.0;
   measOperation[8].out.differencePercent[0..8] := 0.0;
   measOperation[9].out.differencePercent[0..8] := 0.0;
   measOperation[0].out.energyCounter[0] := 4.5557861328125;
   measOperation[0].out.energyCounter[1..8] := 0.0;
   measOperation[1].out.energyCounter[0..8] := 0.0;
   measOperation[2].out.energyCounter[0..8] := 0.0;
   measOperation[3].out.energyCounter[0..8] := 0.0;
   measOperation[4].out.energyCounter[0..8] := 0.0;
   measOperation[5].out.energyCounter[0..8] := 0.0;
   measOperation[6].out.energyCounter[0..8] := 0.0;
   measOperation[7].out.energyCounter[0..8] := 0.0;
   measOperation[8].out.energyCounter[0..8] := 0.0;
   measOperation[9].out.energyCounter[0..8] := 0.0;
   measOperation[0].out.energyCounterTotal := 4.5557861328125;
   measOperation[1..9].out.energyCounterTotal := 0.0;
   measOperation[0..9].out.error := FALSE;
   measOperation[0..9].out.energyPerItem := 0.0;
   measOperation[0].stat.counterLast := 277.473693847656;
   measOperation[1..9].stat.counterLast := 0.0;
   measOperation[0].stat.counterDifference := 277.384918212891;
   measOperation[1..9].stat.counterDifference := 0.0;
   measOperation[0].stat.startEnergyValue[0..8] := 0.0;
   measOperation[1].stat.startEnergyValue[0..8] := 0.0;
   measOperation[2].stat.startEnergyValue[0..8] := 0.0;
   measOperation[3].stat.startEnergyValue[0..8] := 0.0;
   measOperation[4].stat.startEnergyValue[0..8] := 0.0;
   measOperation[5].stat.startEnergyValue[0..8] := 0.0;
   measOperation[6].stat.startEnergyValue[0..8] := 0.0;
   measOperation[7].stat.startEnergyValue[0..8] := 0.0;
   measOperation[8].stat.startEnergyValue[0..8] := 0.0;
   measOperation[9].stat.startEnergyValue[0..8] := 0.0;
   measOperation[0..9].stat.energyCounterIntermediate := 0.0;
   measOperation[0].stat.energyEnPiCalc[0] := 4.555786;
   measOperation[0].stat.energyEnPiCalc[1..8] := 0.0;
   measOperation[1].stat.energyEnPiCalc[0..8] := 0.0;
   measOperation[2].stat.energyEnPiCalc[0..8] := 0.0;
   measOperation[3].stat.energyEnPiCalc[0..8] := 0.0;
   measOperation[4].stat.energyEnPiCalc[0..8] := 0.0;
   measOperation[5].stat.energyEnPiCalc[0..8] := 0.0;
   measOperation[6].stat.energyEnPiCalc[0..8] := 0.0;
   measOperation[7].stat.energyEnPiCalc[0..8] := 0.0;
   measOperation[8].stat.energyEnPiCalc[0..8] := 0.0;
   measOperation[9].stat.energyEnPiCalc[0..8] := 0.0;
   internalData.productiveEnergyStates[0] := FALSE;
   internalData.productiveEnergyStates[1] := TRUE;
   internalData.productiveEnergyStates[2..8] := FALSE;
   internalData.enpiGoals[0..9] := 0.0;
   internalData.enpiResetTrigger := FALSE;
   internalData.enpiResetTime := DTL#1970-01-01-00:00:00;
   internalData.measPointConfiguration.measPointName := '';
   internalData.measPointConfiguration.measPointMedia := '';
   internalData.measPointConfiguration.measPointUnitCounter := '';
   internalData.measPointConfiguration.measPointUnitActual := '';
   internalData.measPointConfiguration.measPointType := 0;
   internalData.measPointConfiguration.measPointType1Overflow := 0.0;
   internalData.measPointConfiguration.measPointType1NormFactor := 0.0;
   internalData.measPointConfiguration.measPointType2RawLow := 0.0;
   internalData.measPointConfiguration.measPointType2RawHigh := 0.0;
   internalData.measPointConfiguration.measPointType2OutLow := 0.0;
   internalData.measPointConfiguration.measPointType2OutHigh := 0.0;
   internalData.measPointConfiguration.measPointDataSave := FALSE;
   internalData.measPointConfiguration.measPointDataRead := FALSE;
   internalData.measPointConfiguration.measPointInitializationCancel := FALSE;
   internalData.measPointConfiguration.measPointDataWritten := 0;
   internalData.measPointConfiguration.measPointDataIndex := 0;
   internalData.measPointConfiguration.numberMeasPoints := 0;
   internalData.measPointConfiguration.measPointInitialized := FALSE;
   internalData.enmProEnabled := FALSE;
   internalData.enmProData.state := 16#0000;
   internalData.enmProData.error := FALSE;
   internalData.enmProData.save := FALSE;
   internalData.enmProData.abort := FALSE;
   internalData.enmProData.ipAdress[1..4] := 0;
   internalData.enmProData.localPort := 3000;
   internalData.enmProData.remotePort := 3000;
   internalData.enmProData.interfaceId := 64;
   internalData.enmProData.connectionId := 16#000E;
END_DATA_BLOCK

DATA_BLOCK "InstE2MenergyMeterDriver"   // DB56
TITLE = Instanz von FB E2MenergyMeterDrv / Instance of FB E2MenergyMeterDrv
AUTHOR : SICAR
FAMILY : E2M
NAME : E2M_AIEM
VERSION : 2.0
// Energy Meter
// stored: InstanceOfName E2MenergyMeterDrv, InstanceOfType FB
"E2MenergyMeterDrv"
   // VAR_INPUT
   //    id : HW_IO := 0;
   //    firstByteData : Int := 0;
   //    connectionType : Int := 1;
   //    commResourceLimit : Int := 4;
   //    automaticUpdate : Bool := FALSE;
   //    resetMinMax : Bool := FALSE;
   //    resetEnergyCounter : Bool := FALSE;
   //    bitsConnectedHmi : Bool := FALSE;
   //    backupCycleEnCount : Time := T#5S;
   // END_VAR
   // VAR_OUTPUT
   //    timeBetweenUpdate : Time := T#0MS;
   //    timeBetweenUpdateMax : Time := T#0MS;
   //    timeStampMeasValues : DTL := DTL#1970-01-01-00:00:00;
   //    driverData { ExternalAccessible := 'False'; ExternalVisible := 'False'; ExternalWritable := 'False'} : "LSicar_typeEnMeterVisuStruct";
   //    energyCounter { ExternalAccessible := 'False'; ExternalVisible := 'False'; ExternalWritable := 'False'} : "typeEnCounter";
   //    errorCode : DWord := 16#0000_0000;
   //    errorLocation : Word := 16#0000;
   //    timeStampEnCount : DTL := DTL#1970-01-01-00:00:00;
   // END_VAR
   // VAR_IN_OUT
   //    bitsHmi : "typeEnMeterBits";
   //    commResourceCounter : Int := 0;
   // END_VAR
   // VAR
   //    instReadDataRecord { S7_SetPoint := 'True'} : RDREC;
   //    instWriteDataRecord { S7_SetPoint := 'True'} : WRREC;
   //    instEnCountUpdateTimer { S7_SetPoint := 'True'} : TON_TIME;
   //    instTimeMeasurement { S7_SetPoint := 'True'} : TON_TIME;
   //    instWatchdog { S7_SetPoint := 'True'} : TON_TIME;
   //    statInputVariablesOk : Bool := FALSE;
   //    statResetEnCountRequest : Bool := FALSE;
   //    statReadDataRecRequest : Bool := FALSE;
   //    statWriteDataRecRequest : Bool := FALSE;
   //    statRestoreEnergy : Bool := FALSE;
   //    statStartAcyclicHmiOld : Bool := FALSE;
   //    statResetEnergyHmiOld : Bool := FALSE;
   //    statResetEnergyOld : Bool := FALSE;
   //    statResetMinMaxHmiOld : Bool := FALSE;
   //    statResetMinMaxOld : Bool := FALSE;
   //    statRunUpdateTimer : Bool := FALSE;
   //    statWatchdogRun : Bool := FALSE;
   //    statUserDataVariant : Byte := 16#00;
   //    statSmState : Int := 0;
   //    statSmStateNext : Int := 0;
   //    statReadRecIndex : Int := 0;
   //    statReadRecMaxLength : UInt := 0;
   //    statTimetoUpdate : Time := T#0MS;
   //    statVmeasurementValues : "typeEnMeterValues";
   //    statVenergyCounter : "typeEnMeterCounter";
   //    statBitsInternalHmi : "typeEnMeterBits";
   // END_VAR
   // VAR RETAIN
   //    statRestoreEnCountValues : "typeEnMeterRestore";
   // END_VAR
   // VAR
   //    statAuxTimeBetweenUpdateMax { S7_SetPoint := 'True'} : Time := T#0MS;
   //    statErrorCode { ExternalVisible := 'False'} : DWord := 16#0000_0000;
   // END_VAR
BEGIN
   driverData.uL1L2 := 480.6464;
   driverData.uL2L3 := 479.3329;
   driverData.uL3L1 := 482.4024;
   driverData.uL1 := 277.0244;
   driverData.uL2 := 283.0648;
   driverData.uL3 := 272.9026;
   driverData.uL1L2Min := 470.1363;
   driverData.uL2L3Min := 469.0945;
   driverData.uL3L1Min := 472.4617;
   driverData.uL1Min := 271.5103;
   driverData.uL2Min := 277.1332;
   driverData.uL3Min := 267.6445;
   driverData.uL1L2Max := 486.0269;
   driverData.uL2L3Max := 484.8441;
   driverData.uL3L1Max := 487.8807;
   driverData.uL1Max := 280.1993;
   driverData.uL2Max := 286.2231;
   driverData.uL3Max := 276.0547;
   driverData.uPhPhAverage := 480.7939;
   driverData.uPhNaverage := 277.6639;
   driverData.uPhPhAverageMin := 470.5642;
   driverData.uPhNaverageMin := 272.105;
   driverData.uPhPhAverageMax := 486.2456;
   driverData.uPhNaverageMax := 280.8176;
   driverData.iL1 := 0.6297245;
   driverData.iL2 := 0.4116209;
   driverData.iL3 := 0.4021624;
   driverData.iL1Min := 0.5503862;
   driverData.iL2Min := 0.3512777;
   driverData.iL3Min := 0.3410119;
   driverData.iL1Max := 2.701323;
   driverData.iL2Max := 2.376321;
   driverData.iL3Max := 1.768756;
   driverData.iAverage := 0.4811693;
   driverData.iAverageMin := 0.4219982;
   driverData.iAverageMax := 2.194234;
   driverData.f := 59.99327;
   driverData.fMin := 59.9567;
   driverData.fMax := 60.07609;
   driverData.sTotal := 400.7156;
   driverData.sTotalMin := 349.7767;
   driverData.sTotalMax := 1823.43;
   driverData.pTotal := 277.3849;
   driverData.pTotalMin := 220.7085;
   driverData.pTotalMax := 670.0833;
   driverData.qTotal := -19.24654;
   driverData.qTotalMin := -422.0206;
   driverData.qTotalMax := -5.418034;
   driverData.cosL1 := 0.8610036;
   driverData.cosL1Min := 0.3576268;
   driverData.cosL1Max := 0.9157406;
   driverData.cosL2 := 0.5061908;
   driverData.cosL2Min := 0.05827232;
   driverData.cosL2Max := 0.7094496;
   driverData.cosL3 := 0.6214478;
   driverData.cosL3Min := 0.1665398;
   driverData.cosL3Max := 0.7301649;
   driverData.cosAverage := 0.6922238;
   driverData.cosAverageMin := 0.2474333;
   driverData.cosAverageMax := 0.7716895;
   driverData.sL1 := 174.449;
   driverData.sL2 := 116.5154;
   driverData.sL3 := 109.7511;
   driverData.sL1Min := 151.7066;
   driverData.sL2Min := 99.03358;
   driverData.sL3Min := 92.7289;
   driverData.sL1Max := 744.3881;
   driverData.sL2Max := 669.9091;
   driverData.sL3Max := 480.3434;
   driverData.pL1 := 150.2012;
   driverData.pL2 := 58.97903;
   driverData.pL3 := 68.20461;
   driverData.pL1Min := 127.6866;
   driverData.pL2Min := 20.87;
   driverData.pL3Min := 52.5906;
   driverData.pL1Max := 281.8818;
   driverData.pL2Max := 194.1828;
   driverData.pL3Max := 220.8245;
   driverData.qL1 := -4.041785;
   driverData.qL2 := 41.25737;
   driverData.qL3 := -56.46213;
   driverData.qL1Min := -144.4171;
   driverData.qL2Min := -98.00859;
   driverData.qL3Min := -198.8008;
   driverData.qL1Max := 28.71266;
   driverData.qL2Max := 50.3845;
   driverData.qL3Max := -53.43742;
   driverData.eActiveRate1Import := 736796.1;
   driverData.eActiveRate2Import := 0.0;
   driverData.eActiveRate1Export := 0.0002530577;
   driverData.eActiveRate2Export := 0.0;
   driverData.eReactiveRate1Import := 5676.457;
   driverData.eReactiveRate2Import := 0.0;
   driverData.eReactiveRate1Export := 293593.3;
   driverData.eReactiveRate2Export := 0.0;
   driverData.eApparentRate1Import := 1470773.0;
   driverData.eApparentRate2Import := 0.0;
   driverData.rTimeDataEnergy := DTL#1970-01-01-00:00:00;
   driverData.rTimeDataValue := DTL#1970-01-01-00:00:00;
   driverData.uPhPhMod := 16#0000;
   driverData.uPhNmod := 16#0000;
   driverData.iMod := 16#0000;
   driverData.sMod := 16#0000;
   driverData.pMod := 16#0000;
   driverData.qMod := 16#0000;
   driverData.eMod := 16#0000;
   driverData.fMod := 16#0000;
   driverData.cosMod := 16#0000;
   driverData.calculateValue1 := 16#0000;
   driverData.calculateValue2 := 16#0000;
   driverData.calculateValue3 := 16#0000;
   driverData.calculateValue4 := 16#0000;
   driverData.calculateValue5 := 16#0000;
   driverData.calculateValue6 := 16#0000;
   driverData.energyMeterUnit := 16#0000;
   driverData.restStartAuto := FALSE;
   driverData.readValue := FALSE;
   driverData.connectionType := 0;
   driverData.driverError := 0;
   energyCounter.activeRate1Imp := 0.0;
   energyCounter.activeRate1Exp := 0.0;
   energyCounter.activeRate2Imp := 0.0;
   energyCounter.activeRate2Exp := 0.0;
   energyCounter.reactiveRate1Imp := 0.0;
   energyCounter.reactiveRate1Exp := 0.0;
   energyCounter.reactiveRate2Imp := 0.0;
   energyCounter.reactiveRate2Exp := 0.0;
   energyCounter.apparentRate1Imp := 0.0;
   energyCounter.apparentRate2Imp := 0.0;
   instReadDataRecord.REQ := FALSE;
   instReadDataRecord.ID := 0;
   instReadDataRecord.INDEX := 0;
   instReadDataRecord.MLEN := 0;
   instReadDataRecord.VALID := FALSE;
   instReadDataRecord.BUSY := FALSE;
   instReadDataRecord.ERROR := FALSE;
   instReadDataRecord.STATUS := 16#0000_0000;
   instReadDataRecord.LEN := 0;
   instWriteDataRecord.REQ := FALSE;
   instWriteDataRecord.ID := 0;
   instWriteDataRecord.INDEX := 0;
   instWriteDataRecord.LEN := 0;
   instWriteDataRecord.DONE := FALSE;
   instWriteDataRecord.BUSY := FALSE;
   instWriteDataRecord.ERROR := FALSE;
   instWriteDataRecord.STATUS := 16#0000_0000;
   instEnCountUpdateTimer.PT := T#0MS;
   instEnCountUpdateTimer.IN := FALSE;
   instTimeMeasurement.PT := T#0MS;
   instTimeMeasurement.IN := FALSE;
   instWatchdog.PT := T#0MS;
   instWatchdog.IN := FALSE;
   statVmeasurementValues.dataRecordVersion := 16#00;
   statVmeasurementValues.reserved := 16#00;
   statVmeasurementValues.voltageL1N := 0.0;
   statVmeasurementValues.voltageL2N := 0.0;
   statVmeasurementValues.voltageL3N := 0.0;
   statVmeasurementValues.voltageL1L2 := 0.0;
   statVmeasurementValues.voltageL2L3 := 0.0;
   statVmeasurementValues.voltageL3L1 := 0.0;
   statVmeasurementValues.currentL1 := 0.0;
   statVmeasurementValues.currentL2 := 0.0;
   statVmeasurementValues.currentL3 := 0.0;
   statVmeasurementValues.powerFactorL1 := 0.0;
   statVmeasurementValues.powerFactorL2 := 0.0;
   statVmeasurementValues.powerFactorL3 := 0.0;
   statVmeasurementValues.powerFactorOverall := 0.0;
   statVmeasurementValues.frequency := 0.0;
   statVmeasurementValues.voltageSymmetry := 0.0;
   statVmeasurementValues.currentSymmetry := 0.0;
   statVmeasurementValues.apparentPowerL1 := 0.0;
   statVmeasurementValues.apparentPowerL2 := 0.0;
   statVmeasurementValues.apparentPowerL3 := 0.0;
   statVmeasurementValues.apparentPowerOverall := 0.0;
   statVmeasurementValues.reactivePowerL1 := 0.0;
   statVmeasurementValues.reactivePowerL2 := 0.0;
   statVmeasurementValues.reactivePowerL3 := 0.0;
   statVmeasurementValues.reactivePowerOverall := 0.0;
   statVmeasurementValues.effectivePowerL1 := 0.0;
   statVmeasurementValues.effectivePowerL2 := 0.0;
   statVmeasurementValues.effectivePowerL3 := 0.0;
   statVmeasurementValues.effectivePowerOverall := 0.0;
   statVmeasurementValues.phaseAngleL1 := 0.0;
   statVmeasurementValues.phaseAngleL2 := 0.0;
   statVmeasurementValues.phaseAngleL3 := 0.0;
   statVmeasurementValues.appEnOverall32bit := 0.0;
   statVmeasurementValues.reaEnOverall32bit := 0.0;
   statVmeasurementValues.effEnOverall32bit := 0.0;
   statVmeasurementValues.reaEnImport32bit := 0.0;
   statVmeasurementValues.reaEnExport32bit := 0.0;
   statVmeasurementValues.effEnImport32bit := 0.0;
   statVmeasurementValues.effEnExport32bit := 0.0;
   statVmeasurementValues.appEnOverall64bit := 0.0;
   statVmeasurementValues.reaEnOverall64bit := 0.0;
   statVmeasurementValues.effEnOverall64bit := 0.0;
   statVmeasurementValues.reaEnImport64bit := 0.0;
   statVmeasurementValues.reaEnExport64bit := 0.0;
   statVmeasurementValues.effEnImport64bit := 0.0;
   statVmeasurementValues.effEnExport64bit := 0.0;
   statVenergyCounter.dataRecordVersion := 16#00;
   statVenergyCounter.reserved := 16#00;
   statVenergyCounter.controlByte1L1 := 16#00;
   statVenergyCounter.controlByte2L1 := 16#00;
   statVenergyCounter.controlByte1L2 := 16#00;
   statVenergyCounter.controlByte2L2 := 16#00;
   statVenergyCounter.controlByte1L3 := 16#00;
   statVenergyCounter.controlByte2L3 := 16#00;
   statVenergyCounter.effEnImportL1 := 0.0;
   statVenergyCounter.effEnExportL1 := 0.0;
   statVenergyCounter.reaEnImportL1 := 0.0;
   statVenergyCounter.reaEnExportL1 := 0.0;
   statVenergyCounter.appEnL1 := 0.0;
   statVenergyCounter.effEnImportL2 := 0.0;
   statVenergyCounter.effEnExportL2 := 0.0;
   statVenergyCounter.reaEnImportL2 := 0.0;
   statVenergyCounter.reaEnExportL2 := 0.0;
   statVenergyCounter.appEnL2 := 0.0;
   statVenergyCounter.effEnImportL3 := 0.0;
   statVenergyCounter.effEnExportL3 := 0.0;
   statVenergyCounter.reaEnImportL3 := 0.0;
   statVenergyCounter.reaEnExportL3 := 0.0;
   statVenergyCounter.appEnL3 := 0.0;
   statBitsInternalHmi.startAcyclic := FALSE;
   statBitsInternalHmi.startAuto := FALSE;
   statBitsInternalHmi.resetMinMaxData := FALSE;
   statBitsInternalHmi.resetEnergyMeter := FALSE;
   statRestoreEnCountValues.dataRecordVersion := 16#00;
   statRestoreEnCountValues.reserved := 16#00;
   statRestoreEnCountValues.controlByte1L1 := 16#00;
   statRestoreEnCountValues.controlByte2L1 := 16#00;
   statRestoreEnCountValues.controlByte1L2 := 16#00;
   statRestoreEnCountValues.controlByte2L2 := 16#00;
   statRestoreEnCountValues.controlByte1L3 := 16#00;
   statRestoreEnCountValues.controlByte2L3 := 16#00;
   statRestoreEnCountValues.effEnImportL1 := 0.0;
   statRestoreEnCountValues.effEnExportL1 := 0.0;
   statRestoreEnCountValues.reaEnImportL1 := 0.0;
   statRestoreEnCountValues.reaEnExportL1 := 0.0;
   statRestoreEnCountValues.appEnL1 := 0.0;
   statRestoreEnCountValues.effEnImportL2 := 0.0;
   statRestoreEnCountValues.effEnExportL2 := 0.0;
   statRestoreEnCountValues.reaEnImportL2 := 0.0;
   statRestoreEnCountValues.reaEnExportL2 := 0.0;
   statRestoreEnCountValues.appEnL2 := 0.0;
   statRestoreEnCountValues.effEnImportL3 := 0.0;
   statRestoreEnCountValues.effEnExportL3 := 0.0;
   statRestoreEnCountValues.reaEnImportL3 := 0.0;
   statRestoreEnCountValues.reaEnExportL3 := 0.0;
   statRestoreEnCountValues.appEnL3 := 0.0;
END_DATA_BLOCK

